(* CODESYS project CtaAppAbtauung_2.0.0.1.library
   Description: Abtauungs Library der CTA
   Version: 2.0.0.1
   Title: CtaAppAbtauung
   Author: PAD
   DocFormat: reStructuredText
   LanguageModelAttribute: qualified-access-only
   Placeholder: CtaAppAbtauung
   DefaultNamespace: CtaAppAbtauung
   CompiledLibraryCompatibilityVersion: CODESYS V3.5 SP16 Patch 3
   Company: CTA

Project tree, tasks and I/O mapping:
  libraries: CtaSysConfig, 2.0.0.0 (CTA); CtaAppTime, 2.0.0.0 (CTA); VisuSymbols, 4.5.0.0 (System); CtaVisSymbols, 2.0.0.0 (CTA); Standard, 3.5.18.0 (System); CtaAppInfluxLog, 1.0.0.1 (CTA); CtaVisApps, 1.0.0.0 (CTA); CtaVisHelp, 2.0.0.0 (CTA); CtaVisUser, 1.0.0.0 (CTA); CtaAppBasic, 1.0.0.1 (CTA); CtaAppReport, 2.0.0.1 (CTA); CtaAppBmk, 2.0.0.0 (CTA)
  40 Visualizations/
    DIALOG/
      visualisation DIA_ParameterAbtauung
      visualisation DIA_Aussentemperatur
      visualisation DIA_Abtauukriterium
      visualisation DIA_Abtauuanforderung
    ICON/
      visualisation VIS_ABTAUUNG
      visualisation VIS_ABTAUUNG_CheckQuerry
      visualisation VIS_ABTAUUNG_OPEN
    visualisation VIS_AbtauungInfo
    visualisation VIS_AbtauungInfoQuerry
  30 Program Organization Units/
    function block fbAbtauung [ST]: actConfig, actTrendlog, actReport, actState, proAcknowledge, proAvailable, proLockDown, proIsError, proIsWarning, proConfigError, p_scAbtauungHilfsenergie_fbiRepTilLockdown, p_scAbtauungHilfsenergie_fbrTempAbtauEnde, p_scAbtauungHilfsenergie_fbtMaxAbtauungHiEnergie, p_scAbtauungHilfsenergie_fbudiAbtauungenHiEnergie, p_scAbtropfphase_fbtAbtropfzeit, p_scBase_fbtAbtauverzögerung, p_scBase_fbtSperrungAbtauung, p_scBase_fbrMaxAussentemperatur, p_scManual_fbuiManualState, p_scManual_fbxManualResetLockTime, p_scUmluftabtauung_fbrTempAbtauUmluftOk, p_scUmluftabtauung_fbtAbtauzeitUmluft, p_scUmluftabtauung_fbudiAbtauungenUmluft, p_scAbtauukriterium_fbrAbtauukriteriumFix, p_scAbtauukriterium_fbrKorrekturAtLuftkühler, p_scTable_fbr_dT_Leistung1, p_scTable_fbr_dT_Leistung2, p_scTable_fbr_dT_LeistungMax, p_scTable_fbr_dT_LeistungMin, p_scTable_fbrAtLeistung1, p_scTable_fbrAtLeistung2, p_scTable_fbrAtLeistungMax, p_scTable_fbrAtLeistungMin, p_scTable_fbrAtMaxLeistung1, p_scTable_fbrAtMaxLeistung2, p_scTable_fbrAtMaxLeistungMax, p_scTable_fbrAtMaxLeistungMin, p_scTable_fbrAtMinLeistung1, p_scTable_fbrAtMinLeistung2, p_scTable_fbrAtMinLeistungMax, p_scTable_fbrAtMinLeistungMin, p_scTable_fbrAussenaemperaturMax, p_scTable_fbrAussentemperatur, p_scTable_fbrAussentemperaturMin, p_scTable_fbrLeistung1, p_scTable_fbrLeistung2, p_scTable_fbrMaxLeistung, p_scTable_fbrMinLeistung, p_scAussentemperatur_fbtAverageTimeRange, p_scAussentemperatur_fbxAtGemittelt, p_scInfluxDb_fbxEnable, proITF_REPORTMANAGER, prorActAussentemperatur, prorActAustrittstemperatur, prorZieltemperatur, prorActdTAbtauukriterium, prorAbtaukriteriumFix, prorKorrekturfaktorRk, prorActdTRückkühler, prordTAuslegung, prordTLeistung, proxSperrungAktiv, proudiActHilfsenergieAbtauungen, proudiActUmluftAbtaaungen, protSperrzeit, protStartverzögerung, proiStatus, proxAcknowledge, proxDemandAbtauung, proxDemandManualAbtauung, proxGenerelleDemand, proxDemandHilfsenergie, proManualUmluft, proManualHilfsenergie, proManualBeenden, proManualQuitTime, protElapsedHilfsenergie, protElapsedUmluft, protTimeLeftAbtropfen, protTimeLeftHilfsenergie, protTimeLeftUmluft
  00000000-0000-0000-0000-000000000000|D:\CoDeSys\LibrariesV3\trunk\Intern\CAA\CAA Template\3.4.0.0 draft\Placeholder.xml
  00000000-0000-0000-0000-000000000000|D:\CoDeSys\LibrariesV3\trunk\Intern\CAA\CAA Template\3.2.0.3 draft\Prefix.pdf
  00000000-0000-0000-0000-000000000000|D:\CoDeSys\LibrariesV3\trunk\Intern\CAA\CAA Template\3.5.2.0 draft\Placeholder.xml
  20 Structs/
    data type scParameter
    Abtauukriterium/
      Tabelle/
        data type scTable
      data type scAbtauukriterium
    Abtauuanforderung/
      data type scAbtauuanforderung
      Base/
        data type scBase
      Umluftabtauung/
        data type scUmluftabtauung
      AbtauungHilfsenergie/
        data type scAbtauungHilfsenergie
      Abtropfphase/
        data type scAbtropfphase
      Manual/
        data type scManual
    Aussentemperatur/
      data type scAussentemperatur
    Trend/
      data type scTrend
    InfluxDb/
      data type scInfluxDb
  50 Images/
  10 Documenation/
    global variables VersionHistory
    global variables readMe
  21 Interface/
    interface ITF_Abtauung: proAcknowledge, proAvailable, proLockDown, proIsError, proIsWarning, prorActdTAbtauukriterium, prorKorrekturfaktorRk, prorAbtaukriteriumFix, prorActAustrittstemperatur, prorActAussentemperatur, prorZieltemperatur, proxDemandAbtauung, proxDemandManualAbtauung, proxGenerelleDemand, proxDemandHilfsenergie, proxSperrungAktiv, proudiActUmluftAbtaaungen, proudiActHilfsenergieAbtauungen, protSperrzeit, protStartverzögerung, proiStatus, proxAcknowledge, prordTAuslegung, prordTLeistung, prorActdTRückkühler, protElapsedHilfsenergie, protElapsedUmluft, protTimeLeftAbtropfen, protTimeLeftHilfsenergie, protTimeLeftUmluft, p_scAbtauungHilfsenergie_fbudiAbtauungenHiEnergie, p_scAbtauungHilfsenergie_fbrTempAbtauEnde, p_scAbtauungHilfsenergie_fbtMaxAbtauungHiEnergie, p_scAbtauungHilfsenergie_fbiRepTilLockdown, p_scAbtropfphase_fbtAbtropfzeit, p_scBase_fbtAbtauverzögerung, p_scBase_fbtSperrungAbtauung, p_scBase_fbrMaxAussentemperatur, p_scManual_fbxManualResetLockTime, p_scManual_fbuiManualState, p_scUmluftabtauung_fbrTempAbtauUmluftOk, p_scUmluftabtauung_fbtAbtauzeitUmluft, p_scUmluftabtauung_fbudiAbtauungenUmluft, p_scInfluxDb_fbxEnable, p_scAbtauukriterium_fbrAbtauukriteriumFix, p_scAbtauukriterium_fbrKorrekturAtLuftkühler, p_scTable_fbrAtLeistungMax, p_scTable_fbrAtMinLeistung1, p_scTable_fbr_dT_LeistungMin, p_scTable_fbrAtMaxLeistungMax, p_scTable_fbrAtMaxLeistung1, p_scTable_fbr_dT_Leistung2, p_scTable_fbr_dT_Leistung1, p_scTable_fbrAtMaxLeistung2, p_scTable_fbrAussenaemperaturMax, p_scTable_fbrAussentemperaturMin, p_scTable_fbrLeistung2, p_scTable_fbrMinLeistung, p_scTable_fbrAtMinLeistungMax, p_scTable_fbrAtLeistung1, p_scTable_fbrLeistung1, p_scTable_fbrMaxLeistung, p_scTable_fbrAussentemperatur, p_scTable_fbrAtMinLeistungMin, p_scTable_fbrAtMinLeistung2, p_scTable_fbrAtMaxLeistungMin, p_scTable_fbrAtLeistungMin, p_scTable_fbrAtLeistung2, p_scTable_fbr_dT_LeistungMax, p_scAussentemperatur_fbtAverageTimeRange, p_scAussentemperatur_fbxAtGemittelt, proConfigError, proITF_REPORTMANAGER, proManualUmluft, proManualHilfsenergie, proManualBeenden, proManualQuitTime
  11 Library Parameter/
  12 Konstanten/
  60 Textlisten/
    text list Error
    text list Info
    text list Warnung
  13 Globale Variablen/
    global variables GlobalKonstant
  text list GlobalTextList
*)

// 20 Structs/scParameter
TYPE scParameter :
    STRUCT
	// Parameter
	scAbtauuanforderung		:	scAbtauuanforderung;
	scAussentemperatur		:	scAussentemperatur;
	scAbtauukriterium		:	scAbtauukriterium;
	scInfluxDb				:	scInfluxDb;
	scTrend					:	scTrend;
    END_STRUCT
END_TYPE

// 20 Structs/Abtauukriterium/Tabelle/scTable
TYPE scTable :
	STRUCT
		(*Leistungen*)
		fbrMinLeistung				:	CtaSysConfig.fbREAL;
		fbrLeistung1				:	CtaSysConfig.fbREAL;
		fbrLeistung2				:	CtaSysConfig.fbREAL;
		fbrMaxLeistung				:	CtaSysConfig.fbREAL;
		(*Aussentemperaturen*)
		fbrAussentemperaturMin		:	CtaSysConfig.fbREAL;
		fbrAussentemperatur			:	CtaSysConfig.fbREAL;
		fbrAussenaemperaturMax		:	CtaSysConfig.fbREAL;
		(*dT*)
		fbrAtMinLeistungMin			:	CtaSysConfig.fbREAL;
		fbrAtMinLeistung1			:	CtaSysConfig.fbREAL;
		fbrAtMinLeistung2			:	CtaSysConfig.fbREAL;
		fbrAtMinLeistungMax			:	CtaSysConfig.fbREAL;		
		fbrAtLeistungMin			:	CtaSysConfig.fbREAL;
		fbrAtLeistung1				:	CtaSysConfig.fbREAL;
		fbrAtLeistung2				:	CtaSysConfig.fbREAL;
		fbrAtLeistungMax			:	CtaSysConfig.fbREAL;		
		fbrAtMaxLeistungMin			:	CtaSysConfig.fbREAL;
		fbrAtMaxLeistung1			:	CtaSysConfig.fbREAL;
		fbrAtMaxLeistung2			:	CtaSysConfig.fbREAL;
		fbrAtMaxLeistungMax			:	CtaSysConfig.fbREAL;
		(*dT's für Auslösungen*)
		fbr_dT_LeistungMin			:	CtaSysConfig.fbREAL;
		fbr_dT_Leistung1			:	CtaSysConfig.fbREAL;
		fbr_dT_Leistung2			:	CtaSysConfig.fbREAL;
		fbr_dT_LeistungMax			:	CtaSysConfig.fbREAL;
	END_STRUCT
END_TYPE

// 20 Structs/Abtauukriterium/scAbtauukriterium
TYPE scAbtauukriterium :
	STRUCT
		scTable 					:	scTable;
		fbrKorrekturAtLuftkühler	:	CtaSysConfig.fbREAL;		
		fbrAbtauukriteriumFix		:	CtaSysConfig.fbREAL;
	END_STRUCT
END_TYPE

// 20 Structs/Abtauuanforderung/scAbtauuanforderung
TYPE scAbtauuanforderung :
	STRUCT
		scBase					:	scBase;
		scUmluftabtauung		:	scUmluftabtauung;
		scAbtauungHilfsenergie	:	scAbtauungHilfsenergie;
		scAbtropfphase			:	scAbtropfphase;
		scManual				:	scManual;		
	END_STRUCT
END_TYPE

// 20 Structs/Aussentemperatur/scAussentemperatur
TYPE scAussentemperatur :
	STRUCT
		fbxAtGemittelt				:	CtaSysConfig.fbBOOL;
		fbtAverageTimeRange			:	CtaSysConfig.fbTIME;		
	END_STRUCT
END_TYPE

// 20 Structs/Abtauuanforderung/AbtauungHilfsenergie/scAbtauungHilfsenergie
TYPE scAbtauungHilfsenergie :
	STRUCT
		fbrTempAbtauEnde			:	CtaSysConfig.fbREAL;
		fbtMaxAbtauungHiEnergie		:	CtaSysConfig.fbTIME;
		fbiRepTilLockdown			:	CtaSysConfig.fbINT;
		fbudiAbtauungenHiEnergie	:	CtaSysConfig.fbUDINT;
	END_STRUCT
END_TYPE

// 20 Structs/Abtauuanforderung/Abtropfphase/scAbtropfphase
TYPE scAbtropfphase :
	STRUCT
		fbtAbtropfzeit				:	CtaSysConfig.fbTIME;	
	END_STRUCT
END_TYPE

// 20 Structs/Abtauuanforderung/Base/scBase
TYPE scBase :
	STRUCT
		fbtAbtauverzögerung			:	CtaSysConfig.fbTIME;
		fbtSperrungAbtauung			:	CtaSysConfig.fbTIME;
		fbrMaxAussentemperatur		:	CtaSysConfig.fbREAL;	
	END_STRUCT
END_TYPE

// 20 Structs/Abtauuanforderung/Manual/scManual
TYPE scManual :
	STRUCT
		fbxManualResetLockTime	:	CtaSysConfig.fbBOOL;	// Manuelle rücksetzung der Sperrzeit
		fbuiManualState			:	CtaSysConfig.fbUINT;	// 0 = Off, 1 = Umluftabtauung, 2 = Abtauung mit Hilfsenergie , 3 = Abtauung Beenden
	END_STRUCT
END_TYPE

// 20 Structs/Abtauuanforderung/Umluftabtauung/scUmluftabtauung
TYPE scUmluftabtauung :
	STRUCT
		fbrTempAbtauUmluftOk		:	CtaSysConfig.fbREAL;
		fbtAbtauzeitUmluft			:	CtaSysConfig.fbTIME;	
		fbudiAbtauungenUmluft		:	CtaSysConfig.fbUDINT;
	END_STRUCT
END_TYPE

// 20 Structs/Trend/scTrend
TYPE scTrend :
	STRUCT
		fbxEnable	: CtaSysConfig.fbBOOL;
	END_STRUCT
END_TYPE

// 20 Structs/InfluxDb/scInfluxDb
{attribute 'pack_mode' := '1'} 
TYPE scInfluxDb :
    STRUCT
        fbxEnable       :   CtaSysConfig.fbBOOL;
    END_STRUCT
END_TYPE

// 10 Documenation/VersionHistory
(* 

.. image:: ../../Images/CTA_Logo.jpg
   :align: right
   :width: 15% 

**Vorlage**   


============ =========== =========== ============================================
**Date**     **Version** **Author**  **Change**
------------ ----------- ----------- --------------------------------------------
04.03.2021   0.0.0.0     SIS         Vorlage erstellt

============ =========== =========== ============================================


*)
VAR_GLOBAL
    stInfo : STRING:= '0.0.0.0, Vorlage, CTA';
END_VAR

// 10 Documenation/readMe
(*

**ReadMe**
 
 |  **Empfehlung**
 |
 |	Bibliothek CtaAppPid zur implementierung eine PID- Reglers.
 |  Instanzieren Sie den CtaAppPid.fbPid in ihrem Funktionsbaustein oder POU beispielsweise als fbPidX(Komponente)Y. (X = Nr des Reglers; Komponente z.B Pumpe, Antrieb oder Ventilator; Y = Nr der Komponente) 
 |  Deklarieren Sie die Struktur Variable welche als Parameter und zur ansteuerung dienen wie im Code beispiel.
 |  
 |  *Beispiel* 

+-----------------------+---------------------------------------------------------------------------------------------------------------------------------------------------------------------------------------------------------------------------------------------------------------------------------------------------------------------------------------------------------------------------------------------------------------------------------------+
| Beschreibung          |  Code                                                                                                                                                                                                                                                                                                                                                                                                                                 |
+=======================+=======================================================================================================================================================================================================================================================================================================================================================================================================================================+
| Pou oder SmFb         | .. code-block:: codesys                                                                                                                                                                                                                                                                                                                                                                                                               |
|                       |                                                                                                                                                                                                                                                                                                                                                                                                                                       |
|                       |	// Deklaration als VAR im POU oder dem selbsterstellten Funktionsbaustein                                                                                                                                                                                                                                                                                                                                                       	|
|                       |   VAR   																																																																																																								|
|						|	    (*PID*)																																																	 																																																						|
|						|		fbPid1Pumpe1			: CtaAppPid.fbPid;                                                                                                                                                                                                                                                                                                                                                              						|
|                       | 		fbPid2Pumpe1			: CtaAppPid.fbPid;																																																																																														|
| 						|	END_VAR                                                                                                                                                                                                                                                                                                                                                                                                                         	|
+-----------------------+---------------------------------------------------------------------------------------------------------------------------------------------------------------------------------------------------------------------------------------------------------------------------------------------------------------------------------------------------------------------------------------------------------------------------------------+
| Code für Init         | .. code-block:: codesys                                                                                                                                                                                                                                                                                                                                                                                                               |
|                       |   																																																																																																									|
| 						|	// Kopieren des nachfolgenden Codes in eine Action zur Initialisierung der Parameter. Zum Beispiel actParameter.																																																																													|
|                       |	{region "Parameter Pid1Pumpe1"}                                                                                                                                                                                                                                                                                                                                                                                                     |
| 						|		(*Basis*)																																																																																																						|
|						|		fbPid1Pumpe1.scParameter.fbrDeadBand               		(_wertInit :=   0.0									, _minInit :=   	, _maxInit := 		);		//P1 Totband																																																														|
|						|		fbPid1Pumpe1.scParameter.fbrBand						(_wertInit :=   0.0									, _minInit :=   	, _maxInit := 		);		//P2 P- Band																																																														|
|						|		fbPid1Pumpe1.scParameter.fbrTn							(_wertInit :=   0.0									, _minInit :=   	, _maxInit := 		);		//P3 Nachstellzeit																																																													|
|						|		fbPid1Pumpe1.scParameter.fbrTv							(_wertInit :=   0.0									, _minInit :=   	, _maxInit := 		);		//P4 Vorhaltezeit																																																													|
|						|		fbPid1Pumpe1.scParameter.fbxInvert						(_wertInit := FALSE																			);		//P5 Regler Invertierung																																																											|
|						|	{endregion}                                                                                                                                                      																																																																	| 
+-----------------------+---------------------------------------------------------------------------------------------------------------------------------------------------------------------------------------------------------------------------------------------------------------------------------------------------------------------------------------------------------------------------------------------------------------------------------------+
*)                                                                                                                                                                                                                                                                                                                                                                                                                                                               
 VAR_GLOBAL                                                                                                                                                                                                                                                                                                                                                                                                                                                      
    xReadMeDone              :   BOOL;                                                                                                                                                                                                                                                                                                                                                                                                                           
END_VAR

// 13 Globale Variablen/GlobalKonstant
{attribute 'qualified_only'}
VAR_GLOBAL
	stReportTextListError   : CtaAppReport.stReportTextList := 'CtaAppAbtauung.Error';
	stReportTextListWarning : CtaAppReport.stReportTextList := 'CtaAppAbtauung.Warnung';
	stReportTextListInfo    : CtaAppReport.stReportTextList := 'CtaAppAbtauung.Info';	
END_VAR

// 30 Program Organization Units/fbAbtauung
FUNCTION_BLOCK fbAbtauung IMPLEMENTS ITF_Abtauung 
VAR_INPUT
	xRelease					:	BOOL;
	xAcknowledge				:	BOOL;
	xExtLockdown				:	BOOL;
	rActMaschienleistung		:	REAL;	
	rAussentemperatur			:	REAL;
	rAustrittstemperatur		:	REAL;	
	ITF_BMK						:	CtaAppBmk.ITF_BMK;
END_VAR
VAR_OUTPUT
	xDemandUmluft				:	BOOL;
	xDemandHilfsenergie			:	BOOL;
	xDemandAbtropfphase			:	BOOL;	
END_VAR
VAR
	(* Internal States *) 
	scEWI						:	CtaAppReport.scReportNr;
	_xIsWarning					:	BOOL;
	xIsWarning					:	BOOL;
	_xIsError					:	BOOL;
	xIsError					:	BOOL;
	xisEnabled					:	BOOL;

(* Hilfsvariablen *)
	rActdTAuslegung				:	REAL;
	rActdTLeistung				:	REAL;
	rAct_dT_Rückkühler			:	REAL;
	rAct_dT_Abtauukriterium		:	REAL;
	xAbtauen					:	BOOL;
	xAbtauungGestartet			:	BOOL;	
	rAussentemperaturGemittelt	:	REAL;
	xWasHilfsenergie			:	BOOL;
	xWasExternalLockdown		:	BOOL;
	
(* FB's *)
	// Skalierer		
	fbAbtauuScaler1				:	CtaAppBasic.fbscaleVierfach;
	fbAbtauuScaler2				:	CtaAppBasic.fbscaleVierfach;
	fbAbtauuScaler3				:	CtaAppBasic.fbscaleVierfach;	
	fbAbtauuScalerAuslegung		:	CtaAppBasic.fbscaleDreifach;	
	fbSclaerAbtauung			:	CtaAppBasic.fbscaleVierfach;
	// Gemittelte Aussentemperatur	
	fbAverageAt					:	CtaAppBasic.fbAverageAt;
		
(* Bistabile Sr *)
	srSperrungAbtauung			:	Standard.SR;
	
(* Flanken *)
	TRIG_SperrungAbtauung		:	Standard.F_TRIG;
	
(* Timer *)
	// Timer für Startverzögerung einer Abtauung
	TON_AbtauenDemand			:	Standard.TON;
	// Timer für Umluft abtauung	
	TON_AbtauungUmluft			:	Standard.TON;
	// Timer für Maximaldauer der Abtauung hilfsenergie
	TON_MaxAbtauung				:	Standard.TON;
	// Timer für Abtropfphase
	TON_Abtropfphase			:	Standard.TON;
	// Timer für Sperrung der nächsten Abtauung
	TON_SperrungAbtauung		:	Standard.TON;
	
(* Reports *)
	// Manager
	fbReportManager				:	CtaAppReport.fbReportManager;      
    // ForCounter
	difor						:	DINT;
	// Info Array's
	ayInfoReporter				:	ARRAY[1..2] OF CtaAppReport.fbReporter;
	// Info Abtauung mit Umluft gestartet
	xInfoAbtauungUmluft			:	BOOL;
	// Info Abtauung mit Hilfsenergie gestartet
	xInfoAbtauungHilfsenergie	:	BOOL;                                                            
	// Error Array's
	ayErrorReporter				:	ARRAY[1..2] OF CtaAppReport.fbReporter;
	// Error Abtauung zu lange gedauert
	xErrAbtauungToLong			:	BOOL;

(* Trendlogs *)
	fbTrendxAbtauanforderung	:	CtaAppInfluxLog.FB_LOG_NODE_BOOL;
	fbTrendxAbtauungGestartet	:	CtaAppInfluxLog.FB_LOG_NODE_BOOL;
	fbTrenddTAuslegung			:	CtaAppInfluxLog.FB_LOG_NODE_REAL;
	fbTrenddTLeistung			:	CtaAppInfluxLog.FB_LOG_NODE_REAL;
	fbAbtauukriterium			:	CtaAppInfluxLog.FB_LOG_NODE_REAL;
	fbTrendrdTRückkühler		:	CtaAppInfluxLog.FB_LOG_NODE_REAL;
	fbTrendxError				:	CtaAppInfluxLog.FB_LOG_NODE_BOOL;		
	
(* Parameter *)
	scParameter					:	scParameter;
	
(* fbConfigfile *)
	fbConfigFile 				:	CtaSysConfig.fbConfigFile;
	xConfigError				:	BOOL;
	
END_VAR

actConfig();

IF NOT xConfigError THEN

	// Prüfen ob kürzlich eine Abtauung gestartet wurde
	TRIG_SperrungAbtauung(CLK	:=	(( xDemandUmluft OR xDemandHilfsenergie) AND xAcknowledge));
	
	// Abtauung sperren falls getriggert
	srSperrungAbtauung	(SET1	:=	TRIG_SperrungAbtauung.Q,
						 RESET	:= 	TON_SperrungAbtauung.Q	OR scParameter.scAbtauuanforderung.scManual.fbxManualResetLockTime.xValue );
						 
	IF scParameter.scAbtauuanforderung.scManual.fbxManualResetLockTime.xValue THEN
		scParameter.scAbtauuanforderung.scManual.fbxManualResetLockTime.proValue := FALSE;
	END_IF		
		 
	// Abtauung für dauer der Wiedereinschaltverzögerung sperren					
	TON_SperrungAbtauung	(IN		:=	srSperrungAbtauung.Q1,
						 	 PT		:=	scParameter.scAbtauuanforderung.scBase.fbtSperrungAbtauung.tValue);
						 
	// Prüfen der Fraigabe und Start der Abtauverzögerung bei Abtauuanforderung
	IF xRelease AND NOT srSperrungAbtauung.Q1 AND NOT xIsError THEN
		(* Scaler für die kleinste Aussentemperatur*)
		fbAbtauuScaler1			(rInput	:=	rActMaschienleistung		, 
								 x1		:=	scParameter.scAbtauukriterium.scTable.fbrMinLeistung.rValue				, 	// Kleinste Leistungsstufe
								 x2		:=	scParameter.scAbtauukriterium.scTable.fbrLeistung1.rValue				, 	// Mittlere Leistungsstufe 1
								 x3		:=	scParameter.scAbtauukriterium.scTable.fbrLeistung2.rValue				, 	// Mittlere Leistungsstufe 2
								 x4		:=	scParameter.scAbtauukriterium.scTable.fbrMaxLeistung.rValue				, 	// Grösste Leistungsstufe
								 y1		:=	scParameter.scAbtauukriterium.scTable.fbrAtMinLeistungMin.rValue		, 	// dT für kleinsete Leistungsstufe
								 y2		:=	scParameter.scAbtauukriterium.scTable.fbrAtMinLeistung1.rValue			, 	// dT für mittlere Leistungsstufe 1
								 y3		:=	scParameter.scAbtauukriterium.scTable.fbrAtMinLeistung2.rValue			, 	// dT für mittlere Leistungsstufe 2
								 y4		:=	scParameter.scAbtauukriterium.scTable.fbrAtMinLeistungMax.rValue		);	// dT für grösste Leistungsstufe
						
		(*Scaler für die mittlere Aussentemperatu*)	
		fbAbtauuScaler2			(rInput	:=	rActMaschienleistung		, 
								 x1		:=	scParameter.scAbtauukriterium.scTable.fbrMinLeistung.rValue				, 	// Kleinste Leistungsstufe         
								 x2		:=	scParameter.scAbtauukriterium.scTable.fbrLeistung1.rValue				, 	// Mittlere Leistungsstufe 1       
								 x3		:=	scParameter.scAbtauukriterium.scTable.fbrLeistung2.rValue				, 	// Mittlere Leistungsstufe 2       
								 x4		:=	scParameter.scAbtauukriterium.scTable.fbrMaxLeistung.rValue				, 	// Grösste Leistungsstufe          
								 y1		:=	scParameter.scAbtauukriterium.scTable.fbrAtLeistungMin.rValue			, 	// dT für kleinsete Leistungsstufe 
								 y2		:=	scParameter.scAbtauukriterium.scTable.fbrAtLeistung1.rValue				, 	// dT für mittlere Leistungsstufe 1
								 y3		:=	scParameter.scAbtauukriterium.scTable.fbrAtLeistung2.rValue				, 	// dT für mittlere Leistungsstufe 2
								 y4		:=	scParameter.scAbtauukriterium.scTable.fbrAtLeistungMax.rValue			);	// dT für grösste Leistungsstufe   
						 
		(*Scaler für die höchste Aussentemperatu*)
		fbAbtauuScaler3			(rInput	:=	rActMaschienleistung		, 
								 x1		:=	scParameter.scAbtauukriterium.scTable.fbrMinLeistung.rValue				, 	// Kleinste Leistungsstufe         
								 x2		:=	scParameter.scAbtauukriterium.scTable.fbrLeistung1.rValue				, 	// Mittlere Leistungsstufe 1       
								 x3		:=	scParameter.scAbtauukriterium.scTable.fbrLeistung2.rValue				, 	// Mittlere Leistungsstufe 2       
								 x4		:=	scParameter.scAbtauukriterium.scTable.fbrMaxLeistung.rValue				,	// Grösste Leistungsstufe          
								 y1		:=	scParameter.scAbtauukriterium.scTable.fbrAtMaxLeistungMin.rValue		, 	// dT für kleinsete Leistungsstufe 
								 y2		:=	scParameter.scAbtauukriterium.scTable.fbrAtMaxLeistung1.rValue			, 	// dT für mittlere Leistungsstufe 1
								 y3		:=	scParameter.scAbtauukriterium.scTable.fbrAtMaxLeistung2.rValue			, 	// dT für mittlere Leistungsstufe 2
								 y4		:=	scParameter.scAbtauukriterium.scTable.fbrAtMaxLeistungMax.rValue		);	// dT für grösste Leistungsstufe   
		
		(*Scaler für die Abtauung gemäss auslegung*)
		fbAbtauuScalerAuslegung	(rInput	:=	rAussentemperatur,
								 x1		:=	scParameter.scAbtauukriterium.scTable.fbrAussentemperaturMin.rValue		,	// kleinste Aussentemperatur
								 x2		:=	scParameter.scAbtauukriterium.scTable.fbrAussentemperatur.rValue		,	// mittlere Aussentemperatur
								 x3		:=	scParameter.scAbtauukriterium.scTable.fbrAussenaemperaturMax.rValue		,	// grösste Aussentemperatur
								 y1		:=	LIMIT(scParameter.scAbtauukriterium.scTable.fbrAtMinLeistungMin.rValue	,fbAbtauuScaler1.rOutput,	scParameter.scAbtauukriterium.scTable.fbrAtMinLeistungMax.rValue	),
								 y2		:=	LIMIT(scParameter.scAbtauukriterium.scTable.fbrAtLeistungMin.rValue		,fbAbtauuScaler2.rOutput,	scParameter.scAbtauukriterium.scTable.fbrAtLeistungMax.rValue		),
								 y3		:=	LIMIT(scParameter.scAbtauukriterium.scTable.fbrAtMaxLeistungMin.rValue	,fbAbtauuScaler2.rOutput,	scParameter.scAbtauukriterium.scTable.fbrAtMaxLeistungMax.rValue	));
		
		rActdTAuslegung := 	fbAbtauuScalerAuslegung.rOutput;
						
		(*Scaler für Abtauug gemäss Leistung*)
		fbSclaerAbtauung		(rInput	:=	rActMaschienleistung													, 
								 x1		:=	scParameter.scAbtauukriterium.scTable.fbrMinLeistung.rValue				, // Kleinste Leistungsstufe   
								 x2		:=	scParameter.scAbtauukriterium.scTable.fbrLeistung1.rValue				, // Mittlere Leistungsstufe 1 
								 x3		:=	scParameter.scAbtauukriterium.scTable.fbrLeistung2.rValue				, // Mittlere Leistungsstufe 2 
								 x4		:=	scParameter.scAbtauukriterium.scTable.fbrMaxLeistung.rValue				, // Grösste Leistungsstufe    
								 y1		:=	scParameter.scAbtauukriterium.scTable.fbr_dT_LeistungMin.rValue			, // dT für kleinsete Leistungsstufe 
								 y2		:=	scParameter.scAbtauukriterium.scTable.fbr_dT_Leistung1.rValue			, // dT für mittlere Leistungsstufe 1
								 y3		:=	scParameter.scAbtauukriterium.scTable.fbr_dT_Leistung2.rValue			, // dT für mittlere Leistungsstufe 2
								 y4		:=	scParameter.scAbtauukriterium.scTable.fbr_dT_LeistungMax.rValue			);// dT für grösste Leistungsstufe   
		
		rActdTLeistung	:=	LIMIT(scParameter.scAbtauukriterium.scTable.fbr_dT_LeistungMin.rValue,fbSclaerAbtauung.rOutput,scParameter.scAbtauukriterium.scTable.fbr_dT_LeistungMax.rValue);
					
		(*Berechnen und Festlegen des Abtaukriteriums*)	
		rAct_dT_Abtauukriterium := SEL	(scParameter.scAbtauukriterium.fbrAbtauukriteriumFix.rValue <> 0,
										 fbAbtauuScalerAuslegung.rOutput + LIMIT(scParameter.scAbtauukriterium.scTable.fbr_dT_LeistungMin.rValue,fbSclaerAbtauung.rOutput,scParameter.scAbtauukriterium.scTable.fbr_dT_LeistungMax.rValue)+scParameter.scAbtauukriterium.fbrKorrekturAtLuftkühler.rValue,
										 scParameter.scAbtauukriterium.fbrAbtauukriteriumFix.rValue) ;
		
		// Aussentemperatur mitteln						 
		fbAverageAt		(rAT := rAussentemperatur);								 
		rAussentemperaturGemittelt := fbAverageAt.GetAverageAT(TimeRange := scParameter.scAussentemperatur.fbtAverageTimeRange.proValue);	
										 
		(*Berechnung des aktuellen dT des Rückkühlers*)							 
		rAct_dT_Rückkühler := SEL(scParameter.scAussentemperatur.fbxAtGemittelt.xValue,rAussentemperatur,MIN(rAussentemperatur,rAussentemperaturGemittelt)) - rAustrittstemperatur;
		
		// Prüfen der Abtauuanforderung und Verzögern des Abtauustarts
		IF rAct_dT_Rückkühler >= rAct_dT_Abtauukriterium THEN
			TON_AbtauenDemand(IN	:=	TRUE									,
							 PT	:=	scParameter.scAbtauuanforderung.scBase.fbtAbtauverzögerung.tValue	,
							 Q	=>	xAbtauen								);
		ELSE
			TON_AbtauenDemand(IN	:= FALSE	);	
			xAbtauen				:= FALSE	 ;
		END_IF	
	ELSE
		TON_AbtauenDemand(IN	:= FALSE	);	
		xAbtauen	 			:= FALSE	 ;
		rAct_dT_Abtauukriterium	:= 0;
		rAct_dT_Rückkühler		:= 0;
	END_IF
	
	// Abtauuanforderung generieren
	IF NOT xIsError THEN
		// Starten einer manuellen Abtauung
		IF scParameter.scAbtauuanforderung.scManual.fbuiManualState.uiValue = 2 THEN
			xDemandHilfsenergie := TRUE;
			scParameter.scAbtauuanforderung.scManual.fbuiManualState.proValue := 0;
		ELSIF scParameter.scAbtauuanforderung.scManual.fbuiManualState.uiValue = 1 THEN
			xDemandUmluft		:= TRUE;
			scParameter.scAbtauuanforderung.scManual.fbuiManualState.proValue := 0;
		ELSE 
			// Starten einer Abtauung gemäss Abtauukriterium
			IF xAbtauen AND rAussentemperatur <= scParameter.scAbtauuanforderung.scBase.fbrMaxAussentemperatur.rValue THEN
				IF rAussentemperatur > scParameter.scAbtauuanforderung.scUmluftabtauung.fbrTempAbtauUmluftOk.rValue THEN
					xDemandUmluft 		:= TRUE;
				ELSE	
					xDemandHilfsenergie := TRUE;
				END_IF		
			END_IF
		END_IF
	END_IF
	
	// Rückmeldung des Programms Abwarten um Timer zu starten
	IF xAcknowledge AND NOT xIsError THEN
		// Prüfen der geforderten Abtauung auf Umluft
		IF xDemandUmluft THEN
			TON_AbtauungUmluft(	IN	:= TRUE,
								PT	:= scParameter.scAbtauuanforderung.scUmluftabtauung.fbtAbtauzeitUmluft.tValue);
								
			IF NOT xAbtauungGestartet THEN				
				scParameter.scAbtauuanforderung.scUmluftabtauung.fbudiAbtauungenUmluft.proValue := scParameter.scAbtauuanforderung.scUmluftabtauung.fbudiAbtauungenUmluft.proValue + 1;
				xAbtauungGestartet := TRUE;
			END_IF	
			
			xInfoAbtauungUmluft		:= TRUE;
			
			IF TON_AbtauungUmluft.Q THEN
				xDemandUmluft 		:= FALSE;
				xAbtauungGestartet 	:= FALSE;
				xInfoAbtauungUmluft	:= FALSE;
			END_IF
			
		// Prüfen der geforderten Abtauung auf Hilfsenergie	
		ELSIF xDemandHilfsenergie THEN	
		
			IF NOT xAbtauungGestartet THEN				
				scParameter.scAbtauuanforderung.scAbtauungHilfsenergie.fbudiAbtauungenHiEnergie.proValue := scParameter.scAbtauuanforderung.scAbtauungHilfsenergie.fbudiAbtauungenHiEnergie.proValue + 1;
				xAbtauungGestartet := TRUE;
			END_IF	
			// Starten der Verzögerung
			TON_MaxAbtauung(IN := TRUE,
							PT := scParameter.scAbtauuanforderung.scAbtauungHilfsenergie.fbtMaxAbtauungHiEnergie.proValue);
				
			xInfoAbtauungHilfsenergie	:= TRUE;   
			xWasHilfsenergie			:= TRUE;
			
			// Wurde die Zieltemperatur erreicht wird Abtauung beendet
			IF 	rAustrittstemperatur >= scParameter.scAbtauuanforderung.scAbtauungHilfsenergie.fbrTempAbtauEnde.rValue THEN
				xDemandHilfsenergie			:= FALSE;
				xAbtauungGestartet  		:= FALSE;
				TON_MaxAbtauung			(IN	:= FALSE);
				xInfoAbtauungHilfsenergie	:= FALSE;
			// Zieltemperatur wird nicht innerhlab der eingestellten Frist erreicht = Error
			ELSIF TON_MaxAbtauung.Q THEN
				xErrAbtauungToLong			:= TRUE;
				xDemandHilfsenergie			:= FALSE;
				xAbtauungGestartet  		:= FALSE;
				TON_MaxAbtauung			(IN	:= FALSE);
				xInfoAbtauungHilfsenergie	:= FALSE;
			END_IF
			
		// Prüfen der geforderten Betriebsart auf Abtropfphase
		ELSIF xDemandAbtropfphase THEN
							
			// Starten der Verzögerung
			TON_Abtropfphase(	IN 	:= TRUE,
								PT 	:= scParameter.scAbtauuanforderung.scAbtropfphase.fbtAbtropfzeit.proValue);
								
			xWasHilfsenergie		:= FALSE;
					
			// Beenden der Abtropfphase						
			IF TON_Abtropfphase.Q THEN
				TON_Abtropfphase (IN	:= FALSE);							
				xDemandAbtropfphase		:= FALSE;	
			END_IF
					
		ELSE
			TON_AbtauungUmluft	(IN	:= FALSE);
			TON_MaxAbtauung		(IN := FALSE);
			TON_Abtropfphase	(IN	:= FALSE);
		END_IF
	ELSIF NOT xAcknowledge AND NOT xIsError THEN
		IF xWasExternalLockdown THEN
			// Zurücketzen der Timer wenn Lockdown von Ausserhalb des FB's kommt.
			TON_AbtauungUmluft	(IN	:= FALSE);
			TON_MaxAbtauung		(IN := FALSE);
			TON_Abtropfphase	(IN	:= FALSE);
			xWasExternalLockdown	:= FALSE;
		ELSE
			IF xWasHilfsenergie THEN
				xDemandAbtropfphase := TRUE;
			END_IF
		END_IF
		
	ELSIF NOT xAcknowledge AND xIsError THEN
		// Auslösung von xIsError durch Abtauung Hilfsenergie - Wurde nicht innerhalb der Frist erricht
		IF  xIsError THEN
			TON_AbtauungUmluft	(IN	:= FALSE);
			TON_MaxAbtauung		(IN := FALSE);
			TON_Abtropfphase	(IN	:= FALSE);			
			xDemandUmluft			:= FALSE;
			xDemandHilfsenergie		:= FALSE;
			xDemandAbtropfphase		:= TRUE;	// Entsprechend wird Abtropfphase nach wie vor angefordert.
			xErrAbtauungToLong		:= FALSE;	// Zurücksetzen des Fehlers
		END_IF
	END_IF
	
	IF scParameter.scAbtauuanforderung.scManual.fbuiManualState.uiValue = 3 THEN
		// Infos zurücksetzen 
		xInfoAbtauungUmluft			:= FALSE;
		xInfoAbtauungHilfsenergie	:= FALSE;
		// Error zurücksetzen
		xErrAbtauungToLong			:= FALSE;
		// Timer Zurücksetzen
		TON_AbtauungUmluft		(IN	:= FALSE);
		TON_MaxAbtauung			(IN := FALSE);
		TON_Abtropfphase		(IN	:= FALSE);
		// Demands zurücksetzen
		xDemandUmluft				:= FALSE;
		xDemandHilfsenergie			:= FALSE;
		xDemandAbtropfphase			:= FALSE;
		xWasExternalLockdown		:= FALSE;
		// Manualstate zurücksetzen
		IF NOT xAcknowledge THEN
			scParameter.scAbtauuanforderung.scManual.fbuiManualState.proValue := 0;
		END_IF
	END_IF	
	
	IF xExtLockdown AND NOT xIsError THEN
		xWasExternalLockdown	:= TRUE;
	END_IF
	
	// Reports
	IF __QUERYINTERFACE(ITF_BMK,ITF_BMK)THEN
		actReport();
	END_IF
ELSE // Im falle eines Configerrors wird alles zurückgesetzt
	xDemandUmluft				:= FALSE;
	xDemandHilfsenergie 		:= FALSE;
	xDemandAbtropfphase			:= FALSE;
	xInfoAbtauungUmluft			:= FALSE;
	xInfoAbtauungHilfsenergie	:= FALSE;
	xErrAbtauungToLong			:= FALSE;
	TON_AbtauungUmluft		(IN	:= FALSE);
	TON_MaxAbtauung			(IN := FALSE);
	TON_Abtropfphase		(IN	:= FALSE);
	xWasExternalLockdown		:= FALSE;
	
	// Konfigurationsfehler
	IF xConfigError THEN
		IF __QUERYINTERFACE(ITF_BMK,ITF_BMK)THEN
			actReport();
		END_IF
	END_IF
END_IF

// Status
actState();

// Trends
IF __QUERYINTERFACE(ITF_BMK,ITF_BMK) THEN
	actTrendlog();
END_IF

ACTION actConfig:
fbConfigFile();

(*ABTAUANFORDERUNG*)
	(*Base*)
	scParameter.scAbtauuanforderung.scBase.fbtAbtauverzögerung						(_usiParaNr :=  1,	itfConfigFb := fbConfigFile, _WertInit:= T#10M, _MinInit := T#00M,_MaxInit := T#60M	);
	scParameter.scAbtauuanforderung.scBase.fbtSperrungAbtauung						(_usiParaNr :=  2,	itfConfigFb := fbConfigFile, _WertInit:= T#30M, _MinInit := T#00M,_MaxInit := T#24H	);
	(*Umluftabtauung*)
	scParameter.scAbtauuanforderung.scUmluftabtauung.fbrTempAbtauUmluftOk			(_usiParaNr :=  3,	itfConfigFb := fbConfigFile, _WertInit:= 12.00, _MinInit := -50.0,_MaxInit :=  50.0	);
	scParameter.scAbtauuanforderung.scUmluftabtauung.fbtAbtauzeitUmluft				(_usiParaNr :=  4,	itfConfigFb := fbConfigFile, _WertInit:= T#30M, _MinInit := T#00M,_MaxInit := T#24H	);
	scParameter.scAbtauuanforderung.scUmluftabtauung.fbudiAbtauungenUmluft			(_usiParaNr :=  5,	itfConfigFb := fbConfigFile, _WertInit:= 00000, 									);
	(*Abtauung Hilfsenergie*)
	scParameter.scAbtauuanforderung.scAbtauungHilfsenergie.fbrTempAbtauEnde			(_usiParaNr :=  6,	itfConfigFb := fbConfigFile, _WertInit:= 10.00, _MinInit := -50.0,_MaxInit :=  50.0	);
	scParameter.scAbtauuanforderung.scAbtauungHilfsenergie.fbtMaxAbtauungHiEnergie	(_usiParaNr :=  7,	itfConfigFb := fbConfigFile, _WertInit:= T#10M, _MinInit := T#00M,_MaxInit := T#24H	);
	scParameter.scAbtauuanforderung.scAbtauungHilfsenergie.fbiRepTilLockdown		(_usiParaNr :=  8,	itfConfigFb := fbConfigFile, _WertInit:= 00003, 									);
	scParameter.scAbtauuanforderung.scAbtauungHilfsenergie.fbudiAbtauungenHiEnergie	(_usiParaNr :=  9,	itfConfigFb := fbConfigFile, _WertInit:= 00000, 									);
	(*Abtropfphase*)
	scParameter.scAbtauuanforderung.scAbtropfphase.fbtAbtropfzeit					(_usiParaNr := 10,	itfConfigFb := fbConfigFile, _WertInit:= T#10M, _MinInit := T#00M,_MaxInit := T#24H	);
	(*Manuell*)
	scParameter.scAbtauuanforderung.scManual.fbuiManualState						(_usiParaNr := 11,	itfConfigFb := fbConfigFile, _WertInit:= 00000, _MinInit := 00000,_MaxInit := 00003	);
(*ABTAUUKRITERIUM*)	
	(*TABLE*)
		(*Tabele Vertikal*)
		scParameter.scAbtauukriterium.scTable.fbrMinLeistung			(_usiParaNr := 12,	itfConfigFb := fbConfigFile, _MinInit :=   0.0,_MaxInit := 100.0);
		scParameter.scAbtauukriterium.scTable.fbrLeistung1				(_usiParaNr := 13,	itfConfigFb := fbConfigFile, _MinInit :=   0.0,_MaxInit := 100.0);
		scParameter.scAbtauukriterium.scTable.fbrLeistung2				(_usiParaNr := 14,	itfConfigFb := fbConfigFile, _MinInit :=   0.0,_MaxInit := 100.0);
		scParameter.scAbtauukriterium.scTable.fbrMaxLeistung			(_usiParaNr := 15,	itfConfigFb := fbConfigFile, _MinInit :=   0.0,_MaxInit := 100.0);
		(*Tabelle Horizontal*)
		scParameter.scAbtauukriterium.scTable.fbrAussentemperaturMin	(_usiParaNr := 16,	itfConfigFb := fbConfigFile, _MinInit := -50.0,_MaxInit :=  50.0);
		scParameter.scAbtauukriterium.scTable.fbrAussentemperatur		(_usiParaNr := 17,	itfConfigFb := fbConfigFile, _MinInit := -50.0,_MaxInit :=  50.0);
		scParameter.scAbtauukriterium.scTable.fbrAussenaemperaturMax	(_usiParaNr := 18,	itfConfigFb := fbConfigFile, _MinInit := -50.0,_MaxInit :=  50.0);
		(*Tabellen Daten*)
		scParameter.scAbtauukriterium.scTable.fbrAtMinLeistungMin		(_usiParaNr := 19,	itfConfigFb := fbConfigFile, _MinInit := -50.0,_MaxInit :=  50.0);
		scParameter.scAbtauukriterium.scTable.fbrAtMinLeistung1			(_usiParaNr := 20,	itfConfigFb := fbConfigFile, _MinInit := -50.0,_MaxInit :=  50.0);
		scParameter.scAbtauukriterium.scTable.fbrAtMinLeistung2			(_usiParaNr := 21,	itfConfigFb := fbConfigFile, _MinInit := -50.0,_MaxInit :=  50.0);
		scParameter.scAbtauukriterium.scTable.fbrAtMinLeistungMax		(_usiParaNr := 22,	itfConfigFb := fbConfigFile, _MinInit := -50.0,_MaxInit :=  50.0);
		scParameter.scAbtauukriterium.scTable.fbrAtLeistungMin			(_usiParaNr := 23,	itfConfigFb := fbConfigFile, _MinInit := -50.0,_MaxInit :=  50.0);
		scParameter.scAbtauukriterium.scTable.fbrAtLeistung1			(_usiParaNr := 24,	itfConfigFb := fbConfigFile, _MinInit := -50.0,_MaxInit :=  50.0);
		scParameter.scAbtauukriterium.scTable.fbrAtLeistung2			(_usiParaNr := 25,	itfConfigFb := fbConfigFile, _MinInit := -50.0,_MaxInit :=  50.0);
		scParameter.scAbtauukriterium.scTable.fbrAtLeistungMax			(_usiParaNr := 26,	itfConfigFb := fbConfigFile, _MinInit := -50.0,_MaxInit :=  50.0);
		scParameter.scAbtauukriterium.scTable.fbrAtMaxLeistungMin		(_usiParaNr := 27,	itfConfigFb := fbConfigFile, _MinInit := -50.0,_MaxInit :=  50.0);
		scParameter.scAbtauukriterium.scTable.fbrAtMaxLeistung1			(_usiParaNr := 28,	itfConfigFb := fbConfigFile, _MinInit := -50.0,_MaxInit :=  50.0);
		scParameter.scAbtauukriterium.scTable.fbrAtMaxLeistung2			(_usiParaNr := 29,	itfConfigFb := fbConfigFile, _MinInit := -50.0,_MaxInit :=  50.0);
		scParameter.scAbtauukriterium.scTable.fbrAtMaxLeistungMax		(_usiParaNr := 30,	itfConfigFb := fbConfigFile, _MinInit := -50.0,_MaxInit :=  50.0);
		(*dT Auslösungen*)
		scParameter.scAbtauukriterium.scTable.fbr_dT_LeistungMin		(_usiParaNr := 31,	itfConfigFb := fbConfigFile, _MinInit :=   0.0,_MaxInit :=  20.0);
		scParameter.scAbtauukriterium.scTable.fbr_dT_Leistung1			(_usiParaNr := 32,	itfConfigFb := fbConfigFile, _MinInit :=   0.0,_MaxInit :=  20.0);
		scParameter.scAbtauukriterium.scTable.fbr_dT_Leistung2			(_usiParaNr := 33,	itfConfigFb := fbConfigFile, _MinInit :=   0.0,_MaxInit :=  20.0);
		scParameter.scAbtauukriterium.scTable.fbr_dT_LeistungMax		(_usiParaNr := 34,	itfConfigFb := fbConfigFile, _MinInit :=   0.0,_MaxInit :=  20.0);
	(* Sonstige *)
	scParameter.scAbtauukriterium.fbrKorrekturAtLuftkühler				(_usiParaNr := 35,	itfConfigFb := fbConfigFile, _MinInit := -20.0,_MaxInit :=  20.0);
	scParameter.scAbtauukriterium.fbrAbtauukriteriumFix					(_usiParaNr := 36,	itfConfigFb := fbConfigFile, _MinInit := -20.0,_MaxInit :=  20.0);
(*AUSSENTEMPERATUR*)
	scParameter.scAussentemperatur.fbxAtGemittelt						(_usiParaNr := 37,	itfConfigFb := fbConfigFile, _WertInit:= FALSE, 									);
	scParameter.scAussentemperatur.fbtAverageTimeRange					(_usiParaNr := 38,	itfConfigFb := fbConfigFile, _WertInit:= T#24H, _MinInit := T#00M,_MaxInit := T#7D	);
(*Influx DB*)
	scParameter.scInfluxDb.fbxEnable									(_usiParaNr := 39,	itfConfigFb := fbConfigFile, _WertInit:=  TRUE, 									);													
(*Trendaufzeichnung*)
	scParameter.scTrend.fbxEnable										(_usiParaNr := 40,	itfConfigFb := fbConfigFile, _WertInit:=  TRUE, 									);													
scParameter.scAbtauuanforderung.scBase.fbrMaxAussentemperatur			(_usiParaNr := 41,	itfConfigFb := fbConfigFile, _MinInit := -20.0,_MaxInit :=  40.0);
END_ACTION

ACTION actTrendlog:
(* Abtauuanforderung *)
fbTrendxAbtauanforderung.ENABLE		:=	scParameter.scTrend.fbxEnable.proValue AND
										scParameter.scInfluxDb.fbxEnable.proValue;
fbTrendxAbtauanforderung.KEY		:=	CONCAT(ITF_BMK.proGetObjectId,'_Abtauuanforderung');
fbTrendxAbtauanforderung.SET_VALUE	:=	xAbtauen;

(* Abtauung gestartet *)
fbTrendxAbtauungGestartet.ENABLE	:=	scParameter.scTrend.fbxEnable.proValue AND
										scParameter.scInfluxDb.fbxEnable.proValue;
fbTrendxAbtauungGestartet.KEY		:=	CONCAT(ITF_BMK.proGetObjectId,'_Abtauung_gestartet');
fbTrendxAbtauungGestartet.SET_VALUE	:=  xAbtauungGestartet;

(* dT aus der Auslegung *)
fbTrenddTAuslegung.ENABLE			:=	scParameter.scTrend.fbxEnable.proValue AND
										scParameter.scInfluxDb.fbxEnable.proValue;
fbTrenddTAuslegung.KEY				:=	CONCAT(ITF_BMK.proGetObjectId,'_dT_Auslegung');
fbTrenddTAuslegung.SET_VALUE		:=  rActdTAuslegung;

(* dT aus der Maschinenleistung *)
fbTrenddTLeistung.ENABLE			:=	scParameter.scTrend.fbxEnable.proValue AND
										scParameter.scInfluxDb.fbxEnable.proValue;
fbTrenddTLeistung.KEY 				:=	CONCAT(ITF_BMK.proGetObjectId,'_dT_Leistung');
fbTrenddTLeistung.SET_VALUE			:=  rActdTLeistung;

(* Abtauukriterium aus Auslegung und Leistung *)
fbAbtauukriterium.ENABLE			:=	scParameter.scTrend.fbxEnable.proValue AND
										scParameter.scInfluxDb.fbxEnable.proValue;
fbAbtauukriterium.KEY 				:=	CONCAT(ITF_BMK.proGetObjectId,'_dT_Abtauukriterium');
fbAbtauukriterium.SET_VALUE			:=  rAct_dT_Abtauukriterium;

(* dT des Rückkühlers At zu Austritt *)
fbTrendrdTRückkühler.ENABLE			:=	scParameter.scTrend.fbxEnable.proValue AND
										scParameter.scInfluxDb.fbxEnable.proValue;
fbTrendrdTRückkühler.KEY 			:=	CONCAT(ITF_BMK.proGetObjectId,'_dT_Rückkühler');
fbTrendrdTRückkühler.SET_VALUE		:=  rAct_dT_Rückkühler;

(* Fehler *)
fbTrendxError.ENABLE				:=	scParameter.scTrend.fbxEnable.proValue AND
										scParameter.scInfluxDb.fbxEnable.proValue;
fbTrendxError.KEY 					:=	CONCAT(ITF_BMK.proGetObjectId,'_Abtauung_xError');
fbTrendxError.SET_VALUE				:=  xIsError;
END_ACTION

ACTION actReport:
(* EWI Manager *)
fbReportManager(	stErrorInitReportTextListIn		:=	ADR(GlobalKonstant.stReportTextListError),
					stWarningInitReportTextListIn	:=	ADR(GlobalKonstant.stReportTextListWarning),
					stInfoInitReportTextListIn		:=	ADR(GlobalKonstant.stReportTextListInfo),
					scReportNr						:=	scEWI);
					
(* Errors *)                        
        (* Meldung Error Abtauung zu lange gedauert *)
        ayErrorReporter[1].proPrio  := 2;
        ayErrorReporter[1].metReport(     		xSetReportIn					:= xErrAbtauungToLong,
												iReportID						:= 1,
												enReportTypeIn					:= CtaAppReport.enReportType.Error,  
												enReportAcknowledgeTypeIn   	:= CtaAppReport.enReportacknowledgeType.RetryN,
												tDelay							:= T#0S, 
												ITF_BMK_IN						:= ITF_BMK,			              
												pstReportTextListIn				:= ADR(GlobalKonstant.stReportTextListError),
												stOptionalReportText		    := '',   
												iRetryTilReportLock 		    := scParameter.scAbtauuanforderung.scAbtauungHilfsenergie.fbiRepTilLockdown.iValue, 
												xResetCount         		    := FALSE,  
												tReset						    := T#24H); 
								
		(* Meldung Configerror *)
        ayErrorReporter[2].proPrio  := 1;
        ayErrorReporter[2].metReport(     		xSetReportIn					:= xConfigError,
												iReportID						:= 2,
												enReportTypeIn					:= CtaAppReport.enReportType.Error,  
												enReportAcknowledgeTypeIn   	:= CtaAppReport.enReportacknowledgeType.Quit,
												tDelay							:= T#0S, 
												ITF_BMK_IN						:= ITF_BMK,			              
												pstReportTextListIn				:= ADR(GlobalKonstant.stReportTextListError),
												stOptionalReportText		    := '',   
												iRetryTilReportLock 		    := 0, 
												xResetCount         		    := FALSE,  
												tReset						    := T#24H);
	
(* Infos *)      
        (* Info Abtauung Umluft gestartet *)      
        ayInfoReporter[1].proPrio := 2;
        ayInfoReporter[1].metReport(			xSetReportIn					:= xInfoAbtauungUmluft AND xAcknowledge,
												iReportID						:= 1,
												enReportTypeIn					:= CtaAppReport.enReportType.Info,  
												enReportAcknowledgeTypeIn   	:= CtaAppReport.enReportAcknowledgeType.Auto,
												tDelay							:= T#0S, 
												ITF_BMK_IN						:= ITF_BMK,			              
												pstReportTextListIn				:= ADR(GlobalKonstant.stReportTextListInfo),
												stOptionalReportText		    := '',   
												iRetryTilReportLock 		    := 0, 
												xResetCount         		    := FALSE,  
												tReset						    := T#24H);  
												
		(* Info Abtauung Hilfsenergie gestartet *)      
        ayInfoReporter[2].proPrio := 2;
        ayInfoReporter[2].metReport(			xSetReportIn					:= xInfoAbtauungHilfsenergie AND xAcknowledge ,
												iReportID						:= 2,
												enReportTypeIn					:= CtaAppReport.enReportType.Info,  
												enReportAcknowledgeTypeIn   	:= CtaAppReport.enReportAcknowledgeType.Auto,
												tDelay							:= T#0S, 
												ITF_BMK_IN						:= ITF_BMK,			              
												pstReportTextListIn				:= ADR(GlobalKonstant.stReportTextListInfo),
												stOptionalReportText		    := '',   
												iRetryTilReportLock 		    := 0, 
												xResetCount         		    := FALSE,  
												tReset						    := T#24H);            
												
(* Sync Reports *)                                         
FOR difor := LOWER_BOUND(ayErrorReporter,1) TO UPPER_BOUND(ayErrorReporter,1) DO
	fbReportManager.metSyncReporter(ayErrorReporter[difor]);	
END_FOR;
FOR difor := LOWER_BOUND(ayInfoReporter,1) TO UPPER_BOUND(ayInfoReporter,1) DO
	fbReportManager.metSyncReporter(ayInfoReporter[difor]);	
END_FOR;
                                                                             
_xIsError   := scEWI.iError <> 0;
_xIsWarning := scEWI.iWarning <> 0;
END_ACTION

ACTION actState:
xisEnabled  :=  NOT xConfigError;
xIsWarning 	:= _xIsWarning;
xIsError	:= _xIsError;
END_ACTION

{attribute 'monitoring' := 'variable'}
PROPERTY proAcknowledge : BOOL
GET
proAcknowledge := NOT proIsError;
END_GET
END_PROPERTY

{attribute 'monitoring' := 'variable'}
PROPERTY proAvailable : BOOL
GET
proAvailable := NOT proIsError;
END_GET
END_PROPERTY

{attribute 'monitoring' := 'variable'}
PROPERTY proLockDown : BOOL
GET
proLockDown := proIsError;
END_GET
END_PROPERTY

PROPERTY proIsError : BOOL
GET
proIsError := xIsError;
END_GET
END_PROPERTY

PROPERTY proIsWarning : BOOL
GET
proIsWarning := xIsWarning;
END_GET
END_PROPERTY

PROPERTY proConfigError : BOOL
GET
proConfigError := xConfigError;
END_GET
END_PROPERTY

PROPERTY p_scAbtauungHilfsenergie_fbiRepTilLockdown : CtaSysConfig.ITF_DATATYPE
GET
p_scAbtauungHilfsenergie_fbiRepTilLockdown := scParameter.scAbtauuanforderung.scAbtauungHilfsenergie.fbiRepTilLockdown;
END_GET
END_PROPERTY

PROPERTY p_scAbtauungHilfsenergie_fbrTempAbtauEnde : CtaSysConfig.ITF_DATATYPE
GET
p_scAbtauungHilfsenergie_fbrTempAbtauEnde := scParameter.scAbtauuanforderung.scAbtauungHilfsenergie.fbrTempAbtauEnde;
END_GET
END_PROPERTY

PROPERTY p_scAbtauungHilfsenergie_fbtMaxAbtauungHiEnergie : CtaSysConfig.ITF_DATATYPE
GET
p_scAbtauungHilfsenergie_fbtMaxAbtauungHiEnergie := scParameter.scAbtauuanforderung.scAbtauungHilfsenergie.fbtMaxAbtauungHiEnergie;
END_GET
END_PROPERTY

PROPERTY p_scAbtauungHilfsenergie_fbudiAbtauungenHiEnergie : CtaSysConfig.ITF_DATATYPE
GET
p_scAbtauungHilfsenergie_fbudiAbtauungenHiEnergie := scParameter.scAbtauuanforderung.scAbtauungHilfsenergie.fbudiAbtauungenHiEnergie;
END_GET
END_PROPERTY

PROPERTY p_scAbtropfphase_fbtAbtropfzeit : CtaSysConfig.ITF_DATATYPE
GET
p_scAbtropfphase_fbtAbtropfzeit := scParameter.scAbtauuanforderung.scAbtropfphase.fbtAbtropfzeit;
END_GET
END_PROPERTY

PROPERTY p_scBase_fbtAbtauverzögerung : CtaSysConfig.ITF_DATATYPE
GET
p_scBase_fbtAbtauverzögerung := scParameter.scAbtauuanforderung.scBase.fbtAbtauverzögerung;
END_GET
END_PROPERTY

PROPERTY p_scBase_fbtSperrungAbtauung : CtaSysConfig.ITF_DATATYPE
GET
p_scBase_fbtSperrungAbtauung := scParameter.scAbtauuanforderung.scBase.fbtSperrungAbtauung;
END_GET
END_PROPERTY

PROPERTY p_scBase_fbrMaxAussentemperatur : CtaSysConfig.ITF_DATATYPE
GET
p_scBase_fbrMaxAussentemperatur := scParameter.scAbtauuanforderung.scBase.fbrMaxAussentemperatur;
END_GET
END_PROPERTY

PROPERTY p_scManual_fbuiManualState : CtaSysConfig.ITF_DATATYPE
GET
p_scManual_fbuiManualState := scParameter.scAbtauuanforderung.scManual.fbuiManualState;
END_GET
END_PROPERTY

PROPERTY p_scManual_fbxManualResetLockTime : CtaSysConfig.ITF_DATATYPE
GET
p_scManual_fbxManualResetLockTime := scParameter.scAbtauuanforderung.scManual.fbxManualResetLockTime;
END_GET
END_PROPERTY

PROPERTY p_scUmluftabtauung_fbrTempAbtauUmluftOk : CtaSysConfig.ITF_DATATYPE
GET
p_scUmluftabtauung_fbrTempAbtauUmluftOk := scParameter.scAbtauuanforderung.scUmluftabtauung.fbrTempAbtauUmluftOk;
END_GET
END_PROPERTY

PROPERTY p_scUmluftabtauung_fbtAbtauzeitUmluft : CtaSysConfig.ITF_DATATYPE
GET
p_scUmluftabtauung_fbtAbtauzeitUmluft := scParameter.scAbtauuanforderung.scUmluftabtauung.fbtAbtauzeitUmluft;
END_GET
END_PROPERTY

PROPERTY p_scUmluftabtauung_fbudiAbtauungenUmluft : CtaSysConfig.ITF_DATATYPE
GET
p_scUmluftabtauung_fbudiAbtauungenUmluft := scParameter.scAbtauuanforderung.scUmluftabtauung.fbudiAbtauungenUmluft;
END_GET
END_PROPERTY

PROPERTY p_scAbtauukriterium_fbrAbtauukriteriumFix : CtaSysConfig.ITF_DATATYPE
GET
p_scAbtauukriterium_fbrAbtauukriteriumFix := scParameter.scAbtauukriterium.fbrAbtauukriteriumFix;
END_GET
END_PROPERTY

PROPERTY p_scAbtauukriterium_fbrKorrekturAtLuftkühler : CtaSysConfig.ITF_DATATYPE
GET
p_scAbtauukriterium_fbrKorrekturAtLuftkühler := scParameter.scAbtauukriterium.fbrKorrekturAtLuftkühler;
END_GET
END_PROPERTY

PROPERTY p_scTable_fbr_dT_Leistung1 : CtaSysConfig.ITF_DATATYPE
GET
p_scTable_fbr_dT_Leistung1 := scParameter.scAbtauukriterium.scTable.fbr_dT_Leistung1;
END_GET
END_PROPERTY

PROPERTY p_scTable_fbr_dT_Leistung2 : CtaSysConfig.ITF_DATATYPE
GET
p_scTable_fbr_dT_Leistung2 := scParameter.scAbtauukriterium.scTable.fbr_dT_Leistung2;
END_GET
END_PROPERTY

PROPERTY p_scTable_fbr_dT_LeistungMax : CtaSysConfig.ITF_DATATYPE
GET
p_scTable_fbr_dT_LeistungMax := scParameter.scAbtauukriterium.scTable.fbr_dT_LeistungMax;
END_GET
END_PROPERTY

PROPERTY p_scTable_fbr_dT_LeistungMin : CtaSysConfig.ITF_DATATYPE
GET
p_scTable_fbr_dT_LeistungMin := scParameter.scAbtauukriterium.scTable.fbr_dT_LeistungMin;
END_GET
END_PROPERTY

PROPERTY p_scTable_fbrAtLeistung1 : CtaSysConfig.ITF_DATATYPE
GET
p_scTable_fbrAtLeistung1 := scParameter.scAbtauukriterium.scTable.fbrAtLeistung1;
END_GET
END_PROPERTY

PROPERTY p_scTable_fbrAtLeistung2 : CtaSysConfig.ITF_DATATYPE
GET
p_scTable_fbrAtLeistung2 := scParameter.scAbtauukriterium.scTable.fbrAtLeistung2;
END_GET
END_PROPERTY

PROPERTY p_scTable_fbrAtLeistungMax : CtaSysConfig.ITF_DATATYPE
GET
p_scTable_fbrAtLeistungMax := scParameter.scAbtauukriterium.scTable.fbrAtLeistungMax;
END_GET
END_PROPERTY

PROPERTY p_scTable_fbrAtLeistungMin : CtaSysConfig.ITF_DATATYPE
GET
p_scTable_fbrAtLeistungMin := scParameter.scAbtauukriterium.scTable.fbrAtLeistungMin;
END_GET
END_PROPERTY

PROPERTY p_scTable_fbrAtMaxLeistung1 : CtaSysConfig.ITF_DATATYPE
GET
p_scTable_fbrAtMaxLeistung1 := scParameter.scAbtauukriterium.scTable.fbrAtMaxLeistung1;
END_GET
END_PROPERTY

PROPERTY p_scTable_fbrAtMaxLeistung2 : CtaSysConfig.ITF_DATATYPE
GET
p_scTable_fbrAtMaxLeistung2 := scParameter.scAbtauukriterium.scTable.fbrAtMaxLeistung2;
END_GET
END_PROPERTY

PROPERTY p_scTable_fbrAtMaxLeistungMax : CtaSysConfig.ITF_DATATYPE
GET
p_scTable_fbrAtMaxLeistungMax := scParameter.scAbtauukriterium.scTable.fbrAtMaxLeistungMax;
END_GET
END_PROPERTY

PROPERTY p_scTable_fbrAtMaxLeistungMin : CtaSysConfig.ITF_DATATYPE
GET
p_scTable_fbrAtMaxLeistungMin := scParameter.scAbtauukriterium.scTable.fbrAtMaxLeistungMin;
END_GET
END_PROPERTY

PROPERTY p_scTable_fbrAtMinLeistung1 : CtaSysConfig.ITF_DATATYPE
GET
p_scTable_fbrAtMinLeistung1 := scParameter.scAbtauukriterium.scTable.fbrAtMinLeistung1;
END_GET
END_PROPERTY

PROPERTY p_scTable_fbrAtMinLeistung2 : CtaSysConfig.ITF_DATATYPE
GET
p_scTable_fbrAtMinLeistung2 := scParameter.scAbtauukriterium.scTable.fbrAtMinLeistung2;
END_GET
END_PROPERTY

PROPERTY p_scTable_fbrAtMinLeistungMax : CtaSysConfig.ITF_DATATYPE
GET
p_scTable_fbrAtMinLeistungMax := scParameter.scAbtauukriterium.scTable.fbrAtMinLeistungMax;
END_GET
END_PROPERTY

PROPERTY p_scTable_fbrAtMinLeistungMin : CtaSysConfig.ITF_DATATYPE
GET
p_scTable_fbrAtMinLeistungMin := scParameter.scAbtauukriterium.scTable.fbrAtMinLeistungMin;
END_GET
END_PROPERTY

PROPERTY p_scTable_fbrAussenaemperaturMax : CtaSysConfig.ITF_DATATYPE
GET
p_scTable_fbrAussenaemperaturMax := scParameter.scAbtauukriterium.scTable.fbrAussenaemperaturMax;
END_GET
END_PROPERTY

PROPERTY p_scTable_fbrAussentemperatur : CtaSysConfig.ITF_DATATYPE
GET
p_scTable_fbrAussentemperatur := scParameter.scAbtauukriterium.scTable.fbrAussentemperatur;
END_GET
END_PROPERTY

PROPERTY p_scTable_fbrAussentemperaturMin : CtaSysConfig.ITF_DATATYPE
GET
p_scTable_fbrAussentemperaturMin := scParameter.scAbtauukriterium.scTable.fbrAussentemperaturMin;
END_GET
END_PROPERTY

PROPERTY p_scTable_fbrLeistung1 : CtaSysConfig.ITF_DATATYPE
GET
p_scTable_fbrLeistung1 := scParameter.scAbtauukriterium.scTable.fbrLeistung1;
END_GET
END_PROPERTY

PROPERTY p_scTable_fbrLeistung2 : CtaSysConfig.ITF_DATATYPE
GET
p_scTable_fbrLeistung2 := scParameter.scAbtauukriterium.scTable.fbrLeistung2;
END_GET
END_PROPERTY

PROPERTY p_scTable_fbrMaxLeistung : CtaSysConfig.ITF_DATATYPE
GET
p_scTable_fbrMaxLeistung := scParameter.scAbtauukriterium.scTable.fbrMaxLeistung;
END_GET
END_PROPERTY

PROPERTY p_scTable_fbrMinLeistung : CtaSysConfig.ITF_DATATYPE
GET
p_scTable_fbrMinLeistung := scParameter.scAbtauukriterium.scTable.fbrMinLeistung;
END_GET
END_PROPERTY

PROPERTY p_scAussentemperatur_fbtAverageTimeRange : CtaSysConfig.ITF_DATATYPE
GET
p_scAussentemperatur_fbtAverageTimeRange := scParameter.scAussentemperatur.fbtAverageTimeRange;
END_GET
END_PROPERTY

PROPERTY p_scAussentemperatur_fbxAtGemittelt : CtaSysConfig.ITF_DATATYPE
GET
p_scAussentemperatur_fbxAtGemittelt := scParameter.scAussentemperatur.fbxAtGemittelt;
END_GET
END_PROPERTY

PROPERTY p_scInfluxDb_fbxEnable : CtaSysConfig.ITF_DATATYPE
GET
p_scInfluxDb_fbxEnable := scParameter.scTrend.fbxEnable;
END_GET
END_PROPERTY

PROPERTY proITF_REPORTMANAGER : CtaAppReport.ITF_REPORTMANAGER
GET
proITF_REPORTMANAGER := fbReportManager;
END_GET
END_PROPERTY

PROPERTY prorActAussentemperatur : REAL
GET
prorActAussentemperatur := SEL(scParameter.scAussentemperatur.fbxAtGemittelt.xValue,rAussentemperatur,MIN(rAussentemperatur,rAussentemperaturGemittelt));
END_GET
END_PROPERTY

PROPERTY prorActAustrittstemperatur : REAL
GET
prorActAustrittstemperatur := rAustrittstemperatur;
END_GET
END_PROPERTY

PROPERTY prorZieltemperatur : REAL
GET
prorZieltemperatur := scParameter.scAbtauuanforderung.scAbtauungHilfsenergie.fbrTempAbtauEnde.proValue;
END_GET
END_PROPERTY

PROPERTY prorActdTAbtauukriterium : REAL
GET
prorActdTAbtauukriterium := rAct_dT_Abtauukriterium;
END_GET
END_PROPERTY

PROPERTY prorAbtaukriteriumFix : REAL
GET
prorAbtaukriteriumFix := scParameter.scAbtauukriterium.fbrAbtauukriteriumFix.rValue;
END_GET
END_PROPERTY

PROPERTY prorKorrekturfaktorRk : REAL
GET
prorKorrekturfaktorRk := scParameter.scAbtauukriterium.fbrKorrekturAtLuftkühler.rValue;
END_GET
END_PROPERTY

PROPERTY prorActdTRückkühler : REAL
GET
prorActdTRückkühler := rAct_dT_Rückkühler;
END_GET
END_PROPERTY

PROPERTY prordTAuslegung : REAL
GET
prordTAuslegung := rActdTAuslegung;
END_GET
END_PROPERTY

PROPERTY prordTLeistung : REAL
GET
prordTLeistung := rActdTLeistung;
END_GET
END_PROPERTY

PROPERTY proxSperrungAktiv : BOOL
GET
proxSperrungAktiv := srSperrungAbtauung.Q1;
END_GET
END_PROPERTY

PROPERTY proudiActHilfsenergieAbtauungen : UDINT
GET
proudiActHilfsenergieAbtauungen := scParameter.scAbtauuanforderung.scAbtauungHilfsenergie.fbudiAbtauungenHiEnergie.proValue;
END_GET
END_PROPERTY

PROPERTY proudiActUmluftAbtaaungen : UDINT
GET
proudiActUmluftAbtaaungen := scParameter.scAbtauuanforderung.scUmluftabtauung.fbudiAbtauungenUmluft.proValue;
END_GET
END_PROPERTY

PROPERTY protSperrzeit : TIME
GET
protSperrzeit := TON_SperrungAbtauung.PT - TON_SperrungAbtauung.ET;
END_GET
END_PROPERTY

PROPERTY protStartverzögerung : TIME
GET
protStartverzögerung := TON_AbtauenDemand.PT - TON_AbtauenDemand.ET;
END_GET
END_PROPERTY

PROPERTY proiStatus : INT
GET
IF xDemandUmluft THEN
	proiStatus := 1;
ELSIF xDemandHilfsenergie THEN
	proiStatus := 2;
ELSIF xDemandAbtropfphase THEN
	proiStatus := 3;
ELSE
	proiStatus := 0;
END_IF
END_GET
END_PROPERTY

PROPERTY proxAcknowledge : BOOL
GET
proxAcknowledge := xAcknowledge;
END_GET
END_PROPERTY

PROPERTY proxDemandAbtauung : BOOL
GET
proxDemandAbtauung := xDemandUmluft OR xDemandHilfsenergie OR xDemandAbtropfphase;
END_GET
END_PROPERTY

PROPERTY proxDemandManualAbtauung : BOOL
GET
proxDemandManualAbtauung := (scParameter.scAbtauuanforderung.scManual.fbuiManualState.uiValue <> 0);
END_GET
END_PROPERTY

PROPERTY proxGenerelleDemand : BOOL
GET
proxGenerelleDemand := TON_AbtauenDemand.IN;
END_GET
END_PROPERTY

PROPERTY proxDemandHilfsenergie : BOOL
GET
proxDemandHilfsenergie := xDemandHilfsenergie;
END_GET
END_PROPERTY

PROPERTY proManualUmluft : BOOL
SET
IF proManualUmluft THEN
	scParameter.scAbtauuanforderung.scManual.fbuiManualState.proValue := 1;
END_IF
END_SET
GET
proManualUmluft := (scParameter.scAbtauuanforderung.scManual.fbuiManualState.proValue = 1);
END_GET
END_PROPERTY

PROPERTY proManualHilfsenergie : BOOL
SET
IF proManualHilfsenergie THEN
	scParameter.scAbtauuanforderung.scManual.fbuiManualState.proValue := 2;
END_IF
END_SET
GET
proManualHilfsenergie := (scParameter.scAbtauuanforderung.scManual.fbuiManualState.proValue = 2);
END_GET
END_PROPERTY

PROPERTY proManualBeenden : BOOL
SET
IF proManualBeenden THEN
	scParameter.scAbtauuanforderung.scManual.fbuiManualState.proValue := 3;
END_IF
END_SET
GET
proManualBeenden := (scParameter.scAbtauuanforderung.scManual.fbuiManualState.proValue = 3);
END_GET
END_PROPERTY

PROPERTY proManualQuitTime : BOOL
SET
IF proManualQuitTime THEN
	scParameter.scAbtauuanforderung.scManual.fbxManualResetLockTime.proValue := TRUE;
END_IF
END_SET
GET
proManualQuitTime := scParameter.scAbtauuanforderung.scManual.fbxManualResetLockTime.proValue;
END_GET
END_PROPERTY

PROPERTY protElapsedHilfsenergie : TIME
GET
protElapsedHilfsenergie := TON_MaxAbtauung.ET;
END_GET
END_PROPERTY

PROPERTY protElapsedUmluft : TIME
GET
protElapsedUmluft := TON_AbtauungUmluft.ET;
END_GET
END_PROPERTY

PROPERTY protTimeLeftAbtropfen : TIME
GET
protTimeLeftAbtropfen := TON_Abtropfphase.PT - TON_Abtropfphase.ET;
END_GET
END_PROPERTY

PROPERTY protTimeLeftHilfsenergie : TIME
GET
protTimeLeftHilfsenergie := TON_MaxAbtauung.PT - TON_MaxAbtauung.ET;
END_GET
END_PROPERTY

PROPERTY protTimeLeftUmluft : TIME
GET
protTimeLeftUmluft := TON_AbtauungUmluft.PT - TON_AbtauungUmluft.ET;
END_GET
END_PROPERTY

END_FUNCTION_BLOCK

// 21 Interface/ITF_Abtauung
INTERFACE ITF_Abtauung EXTENDS __SYSTEM.IQueryInterface

{attribute 'monitoring' := 'variable'}
PROPERTY proAcknowledge : BOOL
GET
END_GET
END_PROPERTY

{attribute 'monitoring' := 'variable'}
PROPERTY proAvailable : BOOL
GET
END_GET
END_PROPERTY

{attribute 'monitoring' := 'variable'}
PROPERTY proLockDown : BOOL
GET
END_GET
END_PROPERTY

PROPERTY proIsError : BOOL
GET
END_GET
END_PROPERTY

PROPERTY proIsWarning : BOOL
GET
END_GET
END_PROPERTY

PROPERTY prorActdTAbtauukriterium : REAL
GET
END_GET
END_PROPERTY

PROPERTY prorKorrekturfaktorRk : REAL
GET
END_GET
END_PROPERTY

PROPERTY prorAbtaukriteriumFix : REAL
GET
END_GET
END_PROPERTY

PROPERTY prorActAustrittstemperatur : REAL
GET
END_GET
END_PROPERTY

PROPERTY prorActAussentemperatur : REAL
GET
END_GET
END_PROPERTY

PROPERTY prorZieltemperatur : REAL
GET
END_GET
END_PROPERTY

PROPERTY proxDemandAbtauung : BOOL
GET
END_GET
END_PROPERTY

PROPERTY proxDemandManualAbtauung : BOOL
GET
END_GET
END_PROPERTY

PROPERTY proxGenerelleDemand : BOOL
GET
END_GET
END_PROPERTY

PROPERTY proxDemandHilfsenergie : BOOL
GET
END_GET
END_PROPERTY

PROPERTY proxSperrungAktiv : BOOL
GET
END_GET
END_PROPERTY

PROPERTY proudiActUmluftAbtaaungen : UDINT
GET
END_GET
END_PROPERTY

PROPERTY proudiActHilfsenergieAbtauungen : UDINT
GET
END_GET
END_PROPERTY

PROPERTY protSperrzeit : TIME
GET
END_GET
END_PROPERTY

PROPERTY protStartverzögerung : TIME
GET
END_GET
END_PROPERTY

PROPERTY proiStatus : INT
GET
END_GET
END_PROPERTY

PROPERTY proxAcknowledge : BOOL
GET
END_GET
END_PROPERTY

PROPERTY prordTAuslegung : REAL
GET
END_GET
END_PROPERTY

PROPERTY prordTLeistung : REAL
GET
END_GET
END_PROPERTY

PROPERTY prorActdTRückkühler : REAL
GET
END_GET
END_PROPERTY

PROPERTY protElapsedHilfsenergie : TIME
GET
END_GET
END_PROPERTY

PROPERTY protElapsedUmluft : TIME
GET
END_GET
END_PROPERTY

PROPERTY protTimeLeftAbtropfen : TIME
GET
END_GET
END_PROPERTY

PROPERTY protTimeLeftHilfsenergie : TIME
GET
END_GET
END_PROPERTY

PROPERTY protTimeLeftUmluft : TIME
GET
END_GET
END_PROPERTY

PROPERTY p_scAbtauungHilfsenergie_fbudiAbtauungenHiEnergie : CtaSysConfig.ITF_DATATYPE
GET
END_GET
END_PROPERTY

PROPERTY p_scAbtauungHilfsenergie_fbrTempAbtauEnde : CtaSysConfig.ITF_DATATYPE
GET
END_GET
END_PROPERTY

PROPERTY p_scAbtauungHilfsenergie_fbtMaxAbtauungHiEnergie : CtaSysConfig.ITF_DATATYPE
GET
END_GET
END_PROPERTY

PROPERTY p_scAbtauungHilfsenergie_fbiRepTilLockdown : CtaSysConfig.ITF_DATATYPE
GET
END_GET
END_PROPERTY

PROPERTY p_scAbtropfphase_fbtAbtropfzeit : CtaSysConfig.ITF_DATATYPE
GET
END_GET
END_PROPERTY

PROPERTY p_scBase_fbtAbtauverzögerung : CtaSysConfig.ITF_DATATYPE
GET
END_GET
END_PROPERTY

PROPERTY p_scBase_fbtSperrungAbtauung : CtaSysConfig.ITF_DATATYPE
GET
END_GET
END_PROPERTY

PROPERTY p_scBase_fbrMaxAussentemperatur : CtaSysConfig.ITF_DATATYPE
GET
END_GET
END_PROPERTY

PROPERTY p_scManual_fbxManualResetLockTime : CtaSysConfig.ITF_DATATYPE
GET
END_GET
END_PROPERTY

PROPERTY p_scManual_fbuiManualState : CtaSysConfig.ITF_DATATYPE
GET
END_GET
END_PROPERTY

PROPERTY p_scUmluftabtauung_fbrTempAbtauUmluftOk : CtaSysConfig.ITF_DATATYPE
GET
END_GET
END_PROPERTY

PROPERTY p_scUmluftabtauung_fbtAbtauzeitUmluft : CtaSysConfig.ITF_DATATYPE
GET
END_GET
END_PROPERTY

PROPERTY p_scUmluftabtauung_fbudiAbtauungenUmluft : CtaSysConfig.ITF_DATATYPE
GET
END_GET
END_PROPERTY

PROPERTY p_scInfluxDb_fbxEnable : CtaSysConfig.ITF_DATATYPE
GET
END_GET
END_PROPERTY

PROPERTY p_scAbtauukriterium_fbrAbtauukriteriumFix : CtaSysConfig.ITF_DATATYPE
GET
END_GET
END_PROPERTY

PROPERTY p_scAbtauukriterium_fbrKorrekturAtLuftkühler : CtaSysConfig.ITF_DATATYPE
GET
END_GET
END_PROPERTY

PROPERTY p_scTable_fbrAtLeistungMax : CtaSysConfig.ITF_DATATYPE
GET
END_GET
END_PROPERTY

PROPERTY p_scTable_fbrAtMinLeistung1 : CtaSysConfig.ITF_DATATYPE
GET
END_GET
END_PROPERTY

PROPERTY p_scTable_fbr_dT_LeistungMin : CtaSysConfig.ITF_DATATYPE
GET
END_GET
END_PROPERTY

PROPERTY p_scTable_fbrAtMaxLeistungMax : CtaSysConfig.ITF_DATATYPE
GET
END_GET
END_PROPERTY

PROPERTY p_scTable_fbrAtMaxLeistung1 : CtaSysConfig.ITF_DATATYPE
GET
END_GET
END_PROPERTY

PROPERTY p_scTable_fbr_dT_Leistung2 : CtaSysConfig.ITF_DATATYPE
GET
END_GET
END_PROPERTY

PROPERTY p_scTable_fbr_dT_Leistung1 : CtaSysConfig.ITF_DATATYPE
GET
END_GET
END_PROPERTY

PROPERTY p_scTable_fbrAtMaxLeistung2 : CtaSysConfig.ITF_DATATYPE
GET
END_GET
END_PROPERTY

PROPERTY p_scTable_fbrAussenaemperaturMax : CtaSysConfig.ITF_DATATYPE
GET
END_GET
END_PROPERTY

PROPERTY p_scTable_fbrAussentemperaturMin : CtaSysConfig.ITF_DATATYPE
GET
END_GET
END_PROPERTY

PROPERTY p_scTable_fbrLeistung2 : CtaSysConfig.ITF_DATATYPE
GET
END_GET
END_PROPERTY

PROPERTY p_scTable_fbrMinLeistung : CtaSysConfig.ITF_DATATYPE
GET
END_GET
END_PROPERTY

PROPERTY p_scTable_fbrAtMinLeistungMax : CtaSysConfig.ITF_DATATYPE
GET
END_GET
END_PROPERTY

PROPERTY p_scTable_fbrAtLeistung1 : CtaSysConfig.ITF_DATATYPE
GET
END_GET
END_PROPERTY

PROPERTY p_scTable_fbrLeistung1 : CtaSysConfig.ITF_DATATYPE
GET
END_GET
END_PROPERTY

PROPERTY p_scTable_fbrMaxLeistung : CtaSysConfig.ITF_DATATYPE
GET
END_GET
END_PROPERTY

PROPERTY p_scTable_fbrAussentemperatur : CtaSysConfig.ITF_DATATYPE
GET
END_GET
END_PROPERTY

PROPERTY p_scTable_fbrAtMinLeistungMin : CtaSysConfig.ITF_DATATYPE
GET
END_GET
END_PROPERTY

PROPERTY p_scTable_fbrAtMinLeistung2 : CtaSysConfig.ITF_DATATYPE
GET
END_GET
END_PROPERTY

PROPERTY p_scTable_fbrAtMaxLeistungMin : CtaSysConfig.ITF_DATATYPE
GET
END_GET
END_PROPERTY

PROPERTY p_scTable_fbrAtLeistungMin : CtaSysConfig.ITF_DATATYPE
GET
END_GET
END_PROPERTY

PROPERTY p_scTable_fbrAtLeistung2 : CtaSysConfig.ITF_DATATYPE
GET
END_GET
END_PROPERTY

PROPERTY p_scTable_fbr_dT_LeistungMax : CtaSysConfig.ITF_DATATYPE
GET
END_GET
END_PROPERTY

PROPERTY p_scAussentemperatur_fbtAverageTimeRange : CtaSysConfig.ITF_DATATYPE
GET
END_GET
END_PROPERTY

PROPERTY p_scAussentemperatur_fbxAtGemittelt : CtaSysConfig.ITF_DATATYPE
GET
END_GET
END_PROPERTY

PROPERTY proConfigError : BOOL
GET
END_GET
END_PROPERTY

{attribute 'hide'} 
PROPERTY INTERNAL proITF_REPORTMANAGER : CtaAppReport.ITF_REPORTMANAGER
GET
END_GET
END_PROPERTY

PROPERTY proManualUmluft : BOOL
SET
END_SET
GET
END_GET
END_PROPERTY

PROPERTY proManualHilfsenergie : BOOL
SET
END_SET
GET
END_GET
END_PROPERTY

PROPERTY proManualBeenden : BOOL
SET
END_SET
GET
END_GET
END_PROPERTY

PROPERTY proManualQuitTime : BOOL
SET
END_SET
GET
END_GET
END_PROPERTY

END_INTERFACE

// 40 Visualizations/DIALOG/DIA_ParameterAbtauung
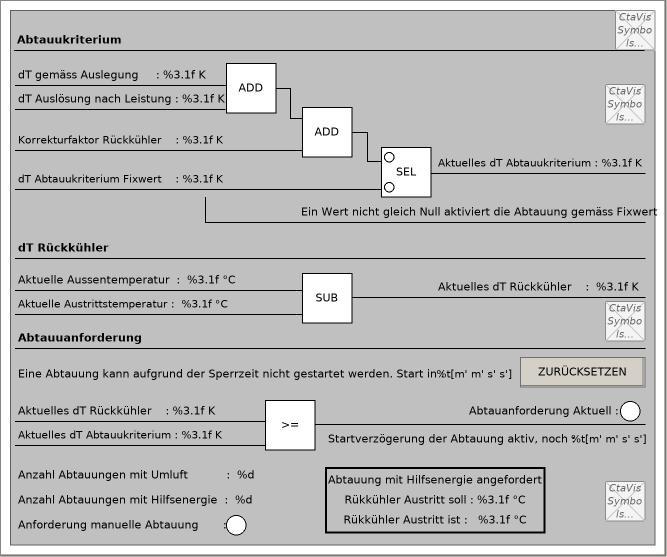
VISUALIZATION DIA_ParameterAbtauung  // 667x557
VAR_IN_OUT
	{attribute 'VAR_IN_OUT_AS_POINTER'}
	ITF_Abtauung_IN		: 	ITF_Abtauung;
END_VAR
    RoundedRectangle (0,0 665x555)
    RoundedRectangle (10,10 645x535)
    Image (615,10 40x40), image: CtaVisSymbols.ImagePool.close_solo_black
        OnMouseClick:  Dialog=Current Dialog, Result=OK, NumpadKeypadSet=True
    Line (15,85) (260,85)
    Line (15,109) (225,109)
    Line (15,150) (310,150)
    Line (15,189) (410,189)
    Line (260,88) (290,88)
    Rectangle (226,63 50x50), "ADD"
    Line (290,88) (290,118)
    Line (290,118) (322,118)
    Line (335,132) (367,132)
    Rectangle (302,107 50x50), "ADD"
    Label (298,202 350x20), "Ein Wert nicht gleich Null aktiviert die Abtauung gemäss Fixwert"
    Line (402,173) (645,173)
    Line (367,161) (399,161)
    Line (367,132) (367,161)
    Rectangle (381,147 50x50), "SEL"
    Ellipse (384,152 10x10), colour toggle: NOT (ITF_Abtauung_IN.prorAbtaukriteriumFix <> 0)
    Ellipse (384,182 10x10), colour toggle: (ITF_Abtauung_IN.prorAbtaukriteriumFix <> 0)
    Rectangle (15,65 210x20), "dT gemäss Auslegung : %3.1f K", text variable: ITF_Abtauung_IN.prordTAuslegung
    Rectangle (15,89 210x20), "dT Auslösung nach Leistung : %3.1f K", text variable: ITF_Abtauung_IN.prordTLeistung
    Rectangle (435,153 210x20), "Aktuelles dT Abtauukriterium : %3.1f K", text variable: ITF_Abtauung_IN.prorActdTAbtauukriterium
    Rectangle (15,130 210x20), "Korrekturfaktor Rückkühler : %3.1f K", text variable: ITF_Abtauung_IN.prorKorrekturfaktorRk
    Rectangle (15,169 210x20), "dT Abtauukriterium Fixwert : %3.1f K", text variable: ITF_Abtauung_IN.prorAbtaukriteriumFix
    Line (205,222) (645,222)
    Line (205,197) (205,222)
    Line (15,258) (645,258)
    Rectangle (15,270 220x20), "Aktuelle Aussentemperatur : %3.1f °C", text variable: ITF_Abtauung_IN.prorActAussentemperatur
    Rectangle (15,294 220x20), "Aktuelle Austrittstemperatur : %3.1f °C", text variable: ITF_Abtauung_IN.prorActAustrittstemperatur
    Rectangle (435,277 210x20), "Aktuelles dT Rückkühler : %3.1f K", text variable: ITF_Abtauung_IN.prorActdTRückkühler
    Line (15,445) (285,445)
    Line (15,421) (285,421)
    Rectangle (15,401 210x20), "Aktuelles dT Rückkühler : %3.1f K", text variable: ITF_Abtauung_IN.prorActdTRückkühler
    Rectangle (15,425 210x20), "Aktuelles dT Abtauukriterium : %3.1f K", text variable: ITF_Abtauung_IN.prorActdTAbtauukriterium
    Line (310,424) (645,424)
    Rectangle (265,400 50x50), ">="
    Label (466,401 150x20), "Abtauanforderung Aktuell :"
    Ellipse (620,401 20x20), colour toggle: ITF_Abtauung_IN.proxGenerelleDemand
    Label (325,429 240x20), "Startverzögerung der Abtauung aktiv, noch :", invisible if: NOT ITF_Abtauung_IN.proxGenerelleDemand OR NOT(ITF_Abtauung_IN.prorActdTRückkühler >= ITF_Abtauung_IN.prorActdTAbtauukriterium)
    Textfield (568,429 80x20), "%t[m' m' s' s']", text variable: ITF_Abtauung_IN.protStartverzögerung, invisible if: NOT ITF_Abtauung_IN.proxGenerelleDemand OR NOT(ITF_Abtauung_IN.prorActdTRückkühler >= ITF_Abtauung_IN.prorActdTAbtauukriterium)
    Rectangle (15,238 220x20), "dT Rückkühler"
    Rectangle (14,30 220x20), "Abtauukriterium"
    Line (14,50) (644,50)
    Rectangle (15,328 220x20), "Abtauuanforderung"
    Line (15,348) (645,348)
    Line (15,290) (310,290)
    Line (15,314) (310,314)
    Line (349,297) (645,297)
    Rectangle (302,273 50x50), "SUB"
    Image (605,84 40x40), image: CtaVisSymbols.ImagePool.gear
        OnMouseClick:  Dialog=DIA_Abtauukriterium, Parameters={ITF_Abtauung_IN: ITF_Abtauung_IN}, Selected={1: }, OpenCentered=True
    Image (605,301 40x40), image: CtaVisSymbols.ImagePool.gear
        OnMouseClick:  Dialog=DIA_Aussentemperatur, Parameters={ITF_Abtauung_IN: ITF_Abtauung_IN}, Selected={1: }, OpenCentered=True
    Label (15,364 411x20), "Eine Abtauung kann aufgrund der Sperrzeit nicht gestartet werden. Start in :", invisible if: NOT ITF_Abtauung_IN.proxSperrungAktiv
    Textfield (430,364 80x20), "%t[m' m' s' s']", text variable: ITF_Abtauung_IN.protSperrzeit, invisible if: NOT ITF_Abtauung_IN.proxSperrungAktiv
    Button (520,357 125x30), "ZURÜCKSETZEN", pressed state: ITF_Abtauung_IN.proManualQuitTime, invisible if: NOT ITF_Abtauung_IN.proxSperrungAktiv
        toggle ITF_Abtauung_IN.proManualQuitTime
        tap ITF_Abtauung_IN.proManualQuitTime
    Image (605,481 40x40), image: CtaVisSymbols.ImagePool.gear
        OnMouseClick:  Dialog=DIA_Abtauuanforderung, Parameters={ITF_Abtauung_IN: ITF_Abtauung_IN}, Selected={1: }, OpenCentered=True
    Label (15,515 250x20), "Anforderung manuelle Abtauung :"
    Ellipse (226,515 20x20), colour toggle: ITF_Abtauung_IN.proxDemandManualAbtauung
    Rectangle (15,465 250x20), "Anzahl Abtauungen mit Umluft : %d", text variable: ITF_Abtauung_IN.proudiActUmluftAbtaaungen
    Rectangle (15,490 250x20), "Anzahl Abtauungen mit Hilfsenergie : %d", text variable: ITF_Abtauung_IN.proudiActHilfsenergieAbtauungen
    Rectangle (325,470 220x20), "Abtauung mit Hilfsenergie angefordert", text variable: ITF_Abtauung_IN.proudiActUmluftAbtaaungen, invisible if: NOT ITF_Abtauung_IN.proxDemandHilfsenergie
    Rectangle (325,490 220x20), "Rükkühler Austritt soll : %3.1f °C", text variable: ITF_Abtauung_IN.prorZieltemperatur, invisible if: NOT ITF_Abtauung_IN.proxDemandHilfsenergie
    Rectangle (325,510 220x20), "Rükkühler Austritt ist : %3.1f °C", text variable: ITF_Abtauung_IN.prorActAustrittstemperatur, invisible if: NOT ITF_Abtauung_IN.proxDemandHilfsenergie
    Rectangle (325,467 220x66), invisible if: NOT ITF_Abtauung_IN.proxDemandHilfsenergie
END_VISUALIZATION

// 40 Visualizations/DIALOG/DIA_Aussentemperatur
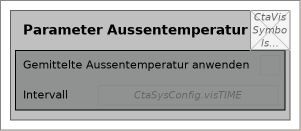
VISUALIZATION DIA_Aussentemperatur  // 301x131
VAR_IN_OUT
	{attribute 'VAR_IN_OUT_AS_POINTER'}
	ITF_Abtauung_IN	:	ITF_Abtauung;
END_VAR
    RoundedRectangle (0,0 300x130)
    RoundedRectangle (10,10 280x110)
    Rectangle (15,50 270x60)
    Label (20,10 350x40), "Parameter Aussentemperatur"
    Image (250,10 40x40), image: CtaVisSymbols.ImagePool.close_solo_black
        OnMouseClick:  Dialog=Current Dialog, Result=OK, NumpadKeypadSet=True
    Label (20,55 230x20), "Gemittelte Aussentemperatur anwenden"
    Frame (260,55 20x20)
        shows CtaSysConfig.visBOOL(visfbBOOLIn := ITF_Abtauung_IN.p_scAussentemperatur_fbxAtGemittelt)
    Label (20,85 60x20), "Intervall"
    Frame (98,85 180x20)
        shows CtaSysConfig.visTIME(visfbTIMEIn := ITF_Abtauung_IN.p_scAussentemperatur_fbtAverageTimeRange)
END_VISUALIZATION

// 40 Visualizations/DIALOG/DIA_Abtauukriterium
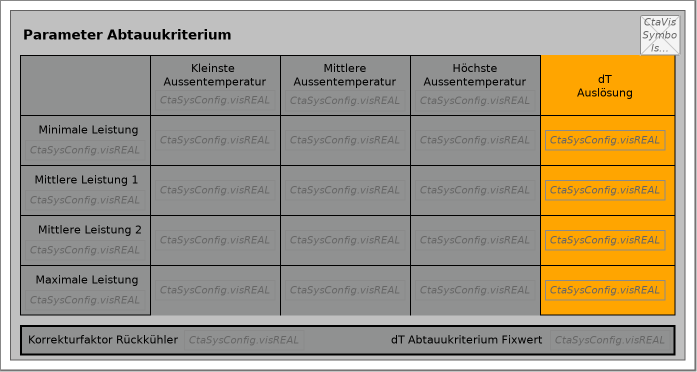
VISUALIZATION DIA_Abtauukriterium  // 697x372
VAR_IN_OUT
	{attribute 'VAR_IN_OUT_AS_POINTER'}
	ITF_Abtauung_IN	:	ITF_Abtauung;
END_VAR
    RoundedRectangle (0,0 695x370)
    RoundedRectangle (10,10 675x350)
    Rectangle (20,325 655x30)
    Rectangle (20,55 655x260)
    Rectangle (151,116 389x199)
    Rectangle (540,55 134x259)
    Rectangle (21,56 130x258)
    Rectangle (21,56 519x60)
    Label (20,15 350x40), "Parameter Abtauukriterium"
    Label (25,330 160x20), "Korrekturfaktor Rückkühler"
    Frame (184,330 120x20)
        shows CtaSysConfig.visREAL(visfbREALIn := ITF_Abtauung_IN.p_scAbtauukriterium_fbrKorrekturAtLuftkühler, stPhysikalischeEinheit := ' K')
    Image (640,15 40x40), image: CtaVisSymbols.ImagePool.close_solo_black
        OnMouseClick:  Dialog=Current Dialog, Result=OK, NumpadKeypadSet=True
    Frame (25,140 120x20)
        shows CtaSysConfig.visREAL(visfbREALIn := ITF_Abtauung_IN.p_scTable_fbrMinLeistung, stPhysikalischeEinheit := ' %')
    Frame (25,190 120x20)
        shows CtaSysConfig.visREAL(visfbREALIn := ITF_Abtauung_IN.p_scTable_fbrLeistung1, stPhysikalischeEinheit := ' %')
    Frame (25,240 120x20)
        shows CtaSysConfig.visREAL(visfbREALIn := ITF_Abtauung_IN.p_scTable_fbrLeistung2, stPhysikalischeEinheit := ' %')
    Frame (25,290 120x20)
        shows CtaSysConfig.visREAL(visfbREALIn := ITF_Abtauung_IN.p_scTable_fbrMaxLeistung, stPhysikalischeEinheit := ' %')
    Label (155,60 120x30), "Kleinste Aussentemperatur"
    Label (25,170 120x20), "Mittlere Leistung 1"
    Label (25,220 120x20), "Mittlere Leistung 2"
    Label (25,270 120x20), "Maximale Leistung"
    Label (285,60 120x30), "Mittlere Aussentemperatur"
    Label (415,60 120x30), "Höchste Aussentemperatur"
    Label (25,120 120x20), "Minimale Leistung"
    Frame (155,90 120x20)
        shows CtaSysConfig.visREAL(visfbREALIn := ITF_Abtauung_IN.p_scTable_fbrAussentemperaturMin, stPhysikalischeEinheit := ' °C')
    Frame (285,90 120x21)
        shows CtaSysConfig.visREAL(visfbREALIn := ITF_Abtauung_IN.p_scTable_fbrAussentemperatur, stPhysikalischeEinheit := ' °C')
    Frame (415,90 120x21)
        shows CtaSysConfig.visREAL(visfbREALIn := ITF_Abtauung_IN.p_scTable_fbrAussenaemperaturMax, stPhysikalischeEinheit := ' °C')
    Line (20,115) (675,115)
    Line (20,165) (675,165)
    Line (20,215) (675,215)
    Line (20,265) (675,265)
    Line (150,55) (150,315)
    Line (280,55) (280,315)
    Line (410,55) (410,315)
    Line (540,55) (540,315)
    Frame (155,130 120x20)
        shows CtaSysConfig.visREAL(visfbREALIn := ITF_Abtauung_IN.p_scTable_fbrAtMinLeistungMin, stPhysikalischeEinheit := ' K')
    Frame (285,130 120x20)
        shows CtaSysConfig.visREAL(visfbREALIn := ITF_Abtauung_IN.p_scTable_fbrAtLeistungMin, stPhysikalischeEinheit := ' K')
    Frame (415,130 120x20)
        shows CtaSysConfig.visREAL(visfbREALIn := ITF_Abtauung_IN.p_scTable_fbrAtMaxLeistungMin, stPhysikalischeEinheit := ' K')
    Frame (545,130 120x20)
        shows CtaSysConfig.visREAL(visfbREALIn := ITF_Abtauung_IN.p_scTable_fbr_dT_LeistungMin, stPhysikalischeEinheit := ' K')
    Frame (155,180 120x20)
        shows CtaSysConfig.visREAL(visfbREALIn := ITF_Abtauung_IN.p_scTable_fbrAtMinLeistung1, stPhysikalischeEinheit := ' K')
    Frame (285,180 120x20)
        shows CtaSysConfig.visREAL(visfbREALIn := ITF_Abtauung_IN.p_scTable_fbrAtLeistung1, stPhysikalischeEinheit := ' K')
    Frame (415,180 120x20)
        shows CtaSysConfig.visREAL(visfbREALIn := ITF_Abtauung_IN.p_scTable_fbrAtMaxLeistung1, stPhysikalischeEinheit := ' K')
    Frame (545,180 120x20)
        shows CtaSysConfig.visREAL(visfbREALIn := ITF_Abtauung_IN.p_scTable_fbr_dT_Leistung1, stPhysikalischeEinheit := ' K')
    Frame (155,230 120x20)
        shows CtaSysConfig.visREAL(visfbREALIn := ITF_Abtauung_IN.p_scTable_fbrAtMinLeistung2, stPhysikalischeEinheit := ' K')
    Frame (285,230 120x20)
        shows CtaSysConfig.visREAL(visfbREALIn := ITF_Abtauung_IN.p_scTable_fbrAtLeistung2, stPhysikalischeEinheit := ' K')
    Frame (415,230 120x20)
        shows CtaSysConfig.visREAL(visfbREALIn := ITF_Abtauung_IN.p_scTable_fbrAtMaxLeistung2, stPhysikalischeEinheit := ' K')
    Frame (545,230 120x20)
        shows CtaSysConfig.visREAL(visfbREALIn := ITF_Abtauung_IN.p_scTable_fbr_dT_Leistung2, stPhysikalischeEinheit := ' K')
    Frame (155,280 120x20)
        shows CtaSysConfig.visREAL(visfbREALIn := ITF_Abtauung_IN.p_scTable_fbrAtMinLeistungMax, stPhysikalischeEinheit := ' K')
    Frame (285,280 120x20)
        shows CtaSysConfig.visREAL(visfbREALIn := ITF_Abtauung_IN.p_scTable_fbrAtLeistungMax, stPhysikalischeEinheit := ' K')
    Frame (415,280 120x20)
        shows CtaSysConfig.visREAL(visfbREALIn := ITF_Abtauung_IN.p_scTable_fbrAtMaxLeistungMax, stPhysikalischeEinheit := ' K')
    Frame (545,280 120x20)
        shows CtaSysConfig.visREAL(visfbREALIn := ITF_Abtauung_IN.p_scTable_fbr_dT_LeistungMax, stPhysikalischeEinheit := ' K')
    Label (545,71 120x30), "dT Auslösung"
    Frame (550,330 120x20)
        shows CtaSysConfig.visREAL(visfbREALIn := ITF_Abtauung_IN.p_scAbtauukriterium_fbrAbtauukriteriumFix, stPhysikalischeEinheit := ' K')
    Label (388,330 160x20), "dT Abtauukriterium Fixwert"
END_VISUALIZATION

// 40 Visualizations/DIALOG/DIA_Abtauuanforderung
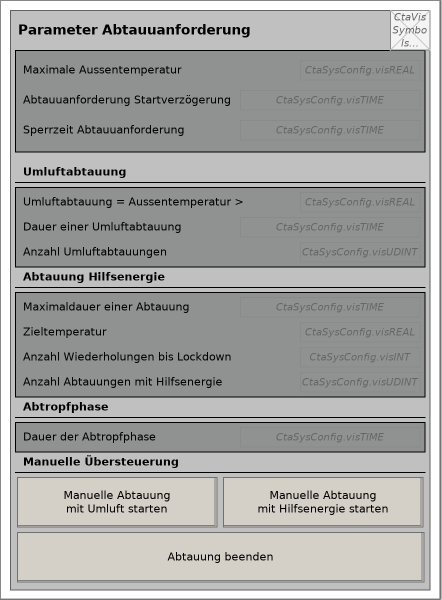
VISUALIZATION DIA_Abtauuanforderung  // 442x600
VAR_IN_OUT
	{attribute 'VAR_IN_OUT_AS_POINTER'}
	ITF_Abtauung_IN		:	ITF_Abtauung;
END_VAR
    RoundedRectangle (0,0 440x600)
    RoundedRectangle (10,10 420x580)
    Rectangle (15,422 410x30)
    Rectangle (15,292 410x105)
    Rectangle (15,187 410x80)
    Rectangle (15,50 410x102)
    Label (15,10 350x40), "Parameter Abtauuanforderung"
    Image (390,10 40x40), image: CtaVisSymbols.ImagePool.close_solo_black
        OnMouseClick:  Dialog=Current Dialog, Result=OK, NumpadKeypadSet=True
    Button (17,532 407x50), "Abtauung beenden", colour toggle: ITF_Abtauung_IN.proManualBeenden, pressed state: ITF_Abtauung_IN.proManualBeenden, invisible if: NOT ITF_Abtauung_IN.proxDemandAbtauung, input disabled if: ITF_Abtauung_IN.proManualBeenden
        toggle ITF_Abtauung_IN.proManualBeenden
    Label (20,90 220x20), "Abtauuanforderung Startverzögerung"
    Frame (240,90 180x20)
        shows CtaSysConfig.visTIME(visfbTIMEIn := ITF_Abtauung_IN.p_scBase_fbtAbtauverzögerung)
    Label (20,120 220x20), "Sperrzeit Abtauuanforderung"
    Frame (240,120 180x20)
        shows CtaSysConfig.visTIME(visfbTIMEIn := ITF_Abtauung_IN.p_scBase_fbtSperrungAbtauung)
    Line (15,182) (425,182)
    Rectangle (20,162 210x20), "Umluftabtauung"
    Label (20,192 220x20), "Umluftabtauung = Aussentemperatur >"
    Frame (300,192 120x20)
        shows CtaSysConfig.visREAL(visfbREALIn := ITF_Abtauung_IN.p_scUmluftabtauung_fbrTempAbtauUmluftOk, stPhysikalischeEinheit := ' °C')
    Frame (240,217 180x20)
        shows CtaSysConfig.visTIME(visfbTIMEIn := ITF_Abtauung_IN.p_scUmluftabtauung_fbtAbtauzeitUmluft)
    Label (20,217 220x20), "Dauer einer Umluftabtauung"
    Label (20,242 220x20), "Anzahl Umluftabtauungen"
    Frame (300,242 120x20)
        shows CtaSysConfig.visUDINT(visfbUDINTIn := ITF_Abtauung_IN.p_scUmluftabtauung_fbudiAbtauungenUmluft)
    Rectangle (20,267 210x20), "Abtauung Hilfsenergie"
    Line (15,287) (425,287)
    Rectangle (20,397 210x20), "Abtropfphase"
    Line (15,417) (425,417)
    Label (20,427 220x20), "Dauer der Abtropfphase"
    Frame (240,427 180x20)
        shows CtaSysConfig.visTIME(visfbTIMEIn := ITF_Abtauung_IN.p_scAbtropfphase_fbtAbtropfzeit)
    Frame (240,297 180x20)
        shows CtaSysConfig.visTIME(visfbTIMEIn := ITF_Abtauung_IN.p_scAbtauungHilfsenergie_fbtMaxAbtauungHiEnergie)
    Label (20,297 220x20), "Maximaldauer einer Abtauung"
    Label (20,372 220x20), "Anzahl Abtauungen mit Hilfsenergie"
    Label (20,347 220x20), "Anzahl Wiederholungen bis Lockdown"
    Button (17,477 200x50), "Manuelle Abtauung mit Umluft starten", colour toggle: ITF_Abtauung_IN.proManualUmluft, pressed state: ITF_Abtauung_IN.proManualUmluft, invisible if: ITF_Abtauung_IN.proxDemandAbtauung, input disabled if: ITF_Abtauung_IN.proxDemandAbtauung
        toggle ITF_Abtauung_IN.proManualUmluft
    Button (223,477 200x50), "Manuelle Abtauung mit Hilfsenergie starten", colour toggle: ITF_Abtauung_IN.proManualHilfsenergie, pressed state: ITF_Abtauung_IN.proManualHilfsenergie, invisible if: ITF_Abtauung_IN.proxDemandAbtauung, input disabled if: ITF_Abtauung_IN.proxDemandAbtauung
        toggle ITF_Abtauung_IN.proManualHilfsenergie
    Rectangle (20,452 200x20), "Manuelle Übersteuerung"
    Line (15,472) (425,472)
    Label (20,322 220x20), "Zieltemperatur"
    Frame (300,372 120x20)
        shows CtaSysConfig.visUDINT(visfbUDINTIn := ITF_Abtauung_IN.p_scAbtauungHilfsenergie_fbudiAbtauungenHiEnergie)
    Frame (300,322 120x20)
        shows CtaSysConfig.visREAL(visfbREALIn := ITF_Abtauung_IN.p_scAbtauungHilfsenergie_fbrTempAbtauEnde, stPhysikalischeEinheit := ' °C')
    Frame (300,347 120x20)
        shows CtaSysConfig.visINT(visfbINTIn := ITF_Abtauung_IN.p_scAbtauungHilfsenergie_fbiRepTilLockdown)
    Label (20,60 220x20), "Maximale Aussentemperatur"
    Frame (300,60 120x20)
        shows CtaSysConfig.visREAL(visfbREALIn := ITF_Abtauung_IN.p_scBase_fbrMaxAussentemperatur, stPhysikalischeEinheit := ' °C')
END_VISUALIZATION

// 40 Visualizations/ICON/VIS_ABTAUUNG
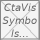
VISUALIZATION VIS_ABTAUUNG  // 40x40
VAR_INPUT
	ITF_Abtauung_IN		: 	ITF_Abtauung;
END_VAR
    Frame (0,0 40x40), invisible if: NOT( __QUERYINTERFACE(ITF_Abtauung_IN,ITF_Abtauung_IN))
        shows VIS_ABTAUUNG_CheckQuerry(ITF_Abtauung_IN := ITF_Abtauung_IN)
END_VISUALIZATION

// 40 Visualizations/ICON/VIS_ABTAUUNG_CheckQuerry
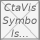
VISUALIZATION VIS_ABTAUUNG_CheckQuerry  // 40x40
VAR_INPUT
	ITF_Abtauung_IN		: 	ITF_Abtauung;
END_VAR
    Frame (0,0 40x40)
        shows VIS_ABTAUUNG_OPEN(ITF_Abtauung_IN := ITF_Abtauung_IN)
END_VISUALIZATION

// 40 Visualizations/ICON/VIS_ABTAUUNG_OPEN
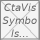
VISUALIZATION VIS_ABTAUUNG_OPEN  // 40x40
VAR_INPUT
	ITF_Abtauung_IN		: 	ITF_Abtauung;
END_VAR
    Image (0,0 40x41), invisible if: NOT __QUERYINTERFACE(ITF_Abtauung_IN,ITF_Abtauung_IN), image: CtaVisSymbols.ImagePool.snowflake_melting_icon
        OnMouseClick:  Dialog=DIA_ParameterAbtauung, Parameters={ITF_Abtauung_IN: ITF_Abtauung_IN}, Selected={0: }, OpenCentered=True
    Rectangle (0,0 40x41)
        OnMouseClick:  Dialog=DIA_ParameterAbtauung, Parameters={ITF_Abtauung_IN: ITF_Abtauung_IN}, Selected={0: }, OpenCentered=True
END_VISUALIZATION

// 40 Visualizations/VIS_AbtauungInfo
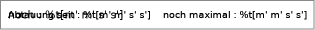
VISUALIZATION VIS_AbtauungInfo  // 315x30
VAR_INPUT
	ITF_Abtauung_IN	: ITF_Abtauung;
END_VAR
    Frame (0,0 315x30), invisible if: NOT( __QUERYINTERFACE(ITF_Abtauung_IN,ITF_Abtauung_IN))
        shows VIS_AbtauungInfoQuerry(ITF_Abtauung_IN := ITF_Abtauung_IN)
END_VISUALIZATION

// 40 Visualizations/VIS_AbtauungInfoQuerry
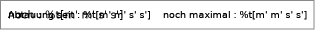
VISUALIZATION VIS_AbtauungInfoQuerry  // 315x30
VAR_INPUT
	ITF_Abtauung_IN	: ITF_Abtauung;
END_VAR
    Textfield (5,5 150x20), "Abtauung seit : %t[m' m' s' s']", text variable: ITF_Abtauung_IN.protElapsedHilfsenergie, invisible if: NOT ITF_Abtauung_IN.proxAcknowledge OR NOT(ITF_Abtauung_IN.proiStatus = 2)
    Textfield (160,5 150x20), "noch maximal : %t[m' m' s' s']", text variable: ITF_Abtauung_IN.protTimeLeftHilfsenergie, invisible if: NOT ITF_Abtauung_IN.proxAcknowledge OR NOT (ITF_Abtauung_IN.proiStatus = 2)
    Textfield (5,5 150x20), "Abtauung seit : %t[m' m' s' s']", text variable: ITF_Abtauung_IN.protElapsedUmluft, invisible if: NOT ITF_Abtauung_IN.proxAcknowledge OR NOT (ITF_Abtauung_IN.proiStatus = 1)
    Textfield (160,5 150x20), "noch maximal : %t[m' m' s' s']", text variable: ITF_Abtauung_IN.protTimeLeftUmluft, invisible if: NOT ITF_Abtauung_IN.proxAcknowledge OR NOT (ITF_Abtauung_IN.proiStatus = 1)
    Textfield (5,5 150x20), "noch : %t[m' m' s' s']", text variable: ITF_Abtauung_IN.protTimeLeftAbtropfen, invisible if: NOT ITF_Abtauung_IN.proxAcknowledge OR NOT (ITF_Abtauung_IN.proiStatus = 3)
END_VISUALIZATION

(* text list Error (id | default | de)
  0 | Keine Meldung Anstehend | Keine Meldung Anstehend
  1 | Abtauung wurde innerhalb der vorgegebenen Frist nicht erreicht | Abtauung wurde innerhalb der vorgegebenen Frist nicht erreicht
  2 | Konfigurationsfehler speichern fehlgeschlagen reboot | Konfigurationsfehler speichern fehlgeschlagen reboot
   |  |  *)

(* text list Info (id | default | de)
  0 | Keine Meldung Anstehend | Keine Meldung Anstehend
  1 | Umluftabtauung wurde gestartet | Umluftabtauung wurde gestartet
  2 | Abtauung mit Hilfsenergie wurde gestartet | Abtauung mit Hilfsenergie wurde gestartet
   |  |  *)

(* text list Warnung (id | default | de)
  3 | Keine Meldung Anstehend | Keine Meldung Anstehend
  4 | Umluftabtauung wurde gestartet | Umluftabtauung wurde gestartet
  5 | Abtauung mit Hilfsenergie wurde gestartet | Abtauung mit Hilfsenergie wurde gestartet
  6 |  | 
   |  |  *)
